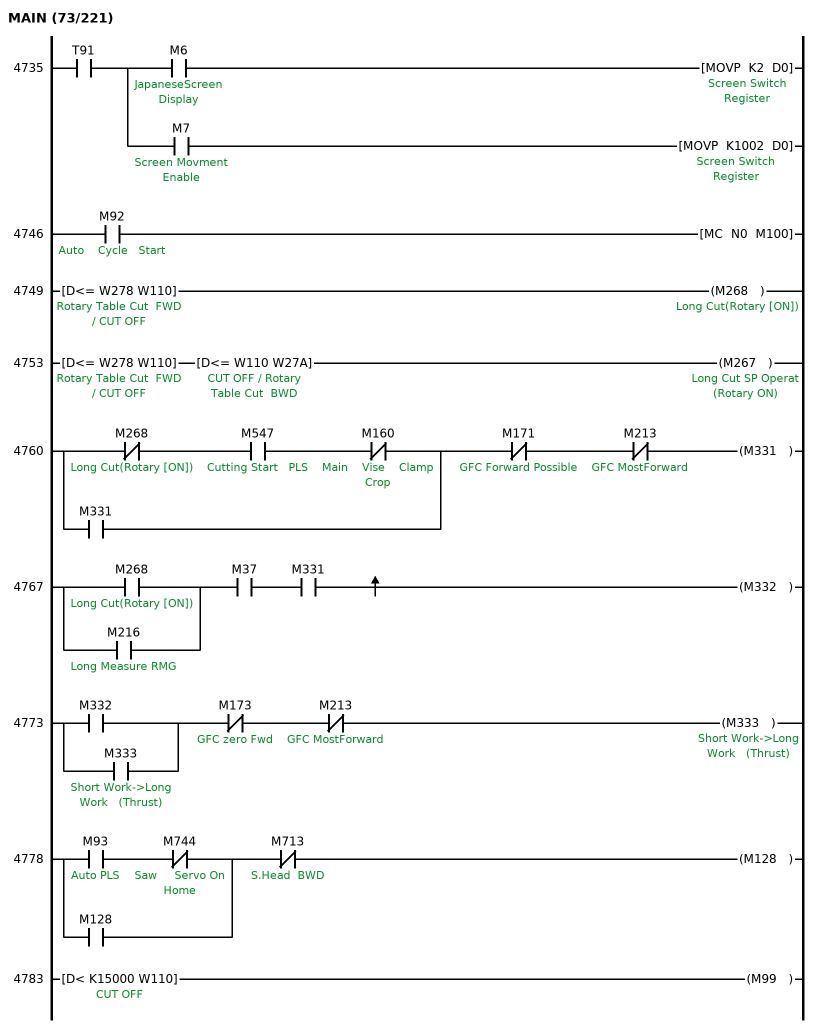
[picture p72: ladder of MAIN, rungs at steps 4735 to 4783]
4735  LD      T91
      MPS
      AND     M6  ; JapaneseScreen Display
      MOVP    K2 D0
      MPP
      AND     M7  ; Screen Movment Enable
      MOVP    K1002 D0
4746  LD      M92  ; Auto    Cycle   Start
      MC      N0 M100
4749  LDD<=   W278 W110  ; Rotary Table Cut  FWD / CUT OFF
      OUT     M268  ; Long Cut(Rotary [ON])
4753  LDD<=   W278 W110  ; Rotary Table Cut  FWD / CUT OFF
      ANDD<=  W110 W27A  ; CUT OFF / Rotary Table Cut  BWD
      OUT     M267  ; Long Cut SP Operat (Rotary ON)
4760  LDI     M268  ; Long Cut(Rotary [ON])
      AND     M547  ; Cutting Start   PLS
      ANI     M160  ; Main    Vise    Clamp   Crop
      OR      M331
      ANI     M171  ; GFC Forward Possible
      ANI     M213  ; GFC MostForward
      OUT     M331
4767  LD      M268  ; Long Cut(Rotary [ON])
      OR      M216  ; Long Measure RMG
      AND     M37
      AND     M331
      MEP
      OUT     M332
4773  LD      M332
      OR      M333  ; Short Work->Long Work   (Thrust)
      ANI     M173  ; GFC zero Fwd
      ANI     M213  ; GFC MostForward
      OUT     M333  ; Short Work->Long Work   (Thrust)
4778  LD      M93  ; Auto PLS
      ANI     M744  ; Saw     Servo On Home
      OR      M128
      ANI     M713  ; S.Head  BWD
      OUT     M128
4783  LDD<    K15000 W110  ; CUT OFF
      OUT     M99
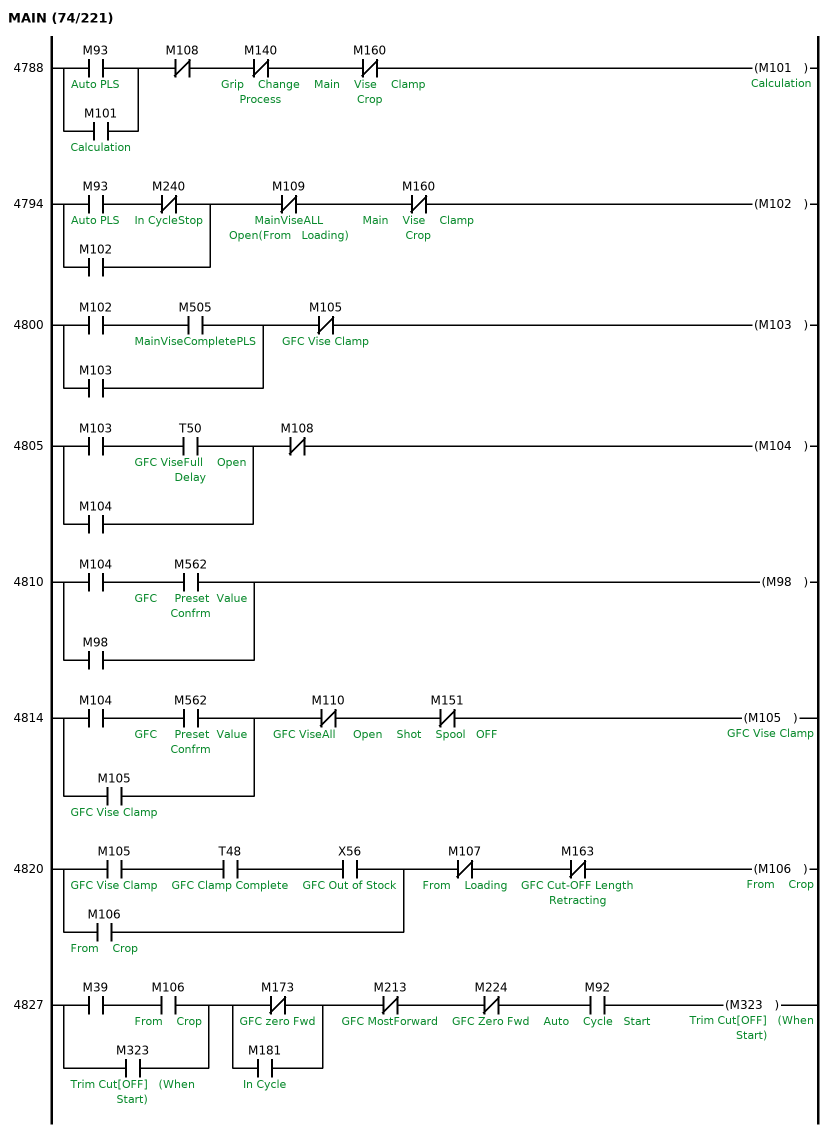
4788  LD      M93  ; Auto PLS
      OR      M101  ; Calculation
      ANI     M108
      ANI     M140  ; Grip    Change  Process
      ANI     M160  ; Main    Vise    Clamp   Crop
      OUT     M101  ; Calculation
4794  LD      M93  ; Auto PLS
      ANI     M240  ; In CycleStop
      OR      M102
      ANI     M109  ; MainViseALL Open(From   Loading)
      ANI     M160  ; Main    Vise    Clamp   Crop
      OUT     M102
4800  LD      M102
      AND     M505  ; MainViseCompletePLS
      OR      M103
      ANI     M105  ; GFC Vise Clamp
      OUT     M103
4805  LD      M103
      AND     T50  ; GFC ViseFull    Open    Delay
      OR      M104
      ANI     M108
      OUT     M104
4810  LD      M104
      AND     M562  ; GFC     Preset  Value   Confrm
      OR      M98
      OUT     M98
4814  LD      M104
      AND     M562  ; GFC     Preset  Value   Confrm
      OR      M105  ; GFC Vise Clamp
      ANI     M110  ; GFC ViseAll     Open
      ANI     M151  ; Shot    Spool   OFF
      OUT     M105  ; GFC Vise Clamp
4820  LD      M105  ; GFC Vise Clamp
      AND     T48  ; GFC Clamp Complete
      AND     X56  ; GFC Out of Stock
      OR      M106  ; From    Crop
      ANI     M107  ; From    Loading
      ANI     M163  ; GFC Cut-OFF Length Retracting
      OUT     M106  ; From    Crop
4827  LD      M39
      AND     M106  ; From    Crop
      OR      M323  ; Trim Cut[OFF]   (When   Start)
      LDI     M173  ; GFC zero Fwd
      OR      M181  ; In Cycle
      ANB
      ANI     M213  ; GFC MostForward
      ANI     M224  ; GFC Zero Fwd
      AND     M92  ; Auto    Cycle   Start
      OUT     M323  ; Trim Cut[OFF]   (When   Start)
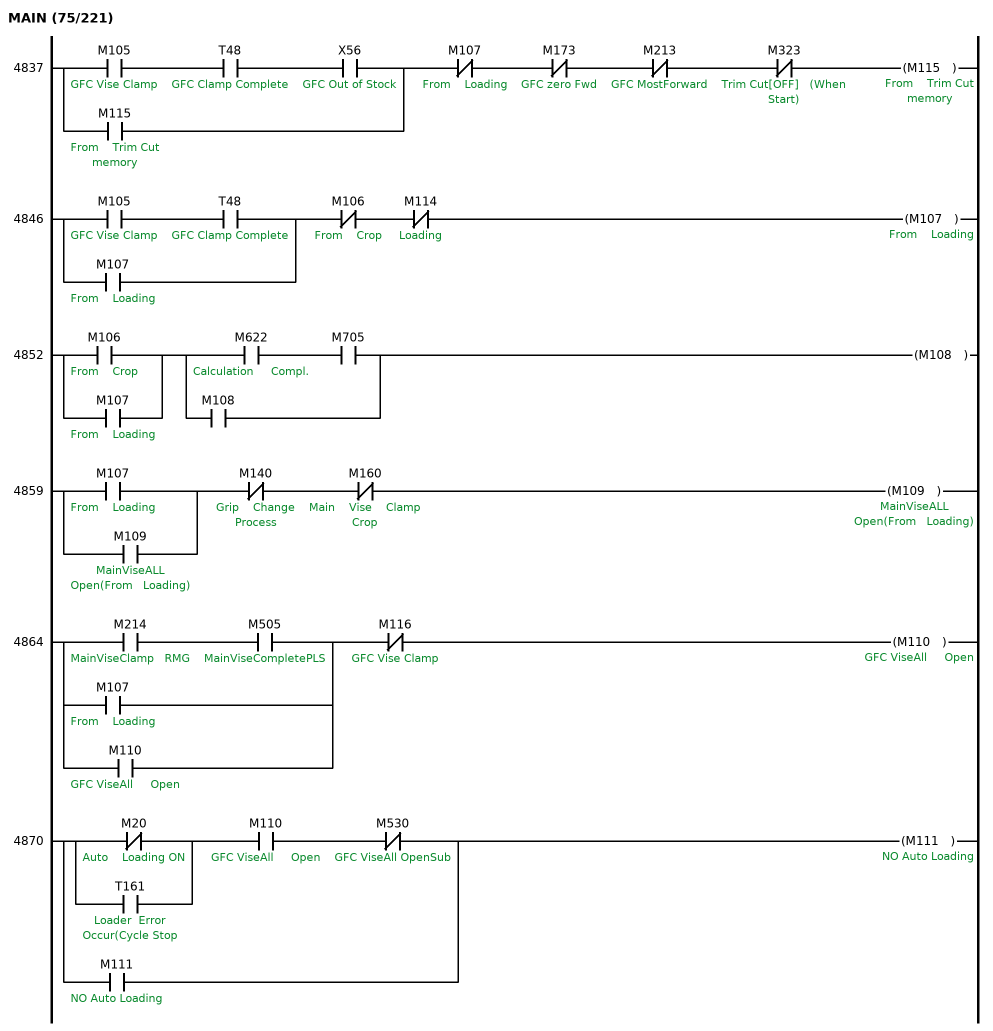
4837  LD      M105  ; GFC Vise Clamp
      AND     T48  ; GFC Clamp Complete
      AND     X56  ; GFC Out of Stock
      OR      M115  ; From    Trim Cut memory
      ANI     M107  ; From    Loading
      ANI     M173  ; GFC zero Fwd
      ANI     M213  ; GFC MostForward
      ANI     M323  ; Trim Cut[OFF]   (When   Start)
      OUT     M115  ; From    Trim Cut memory
4846  LD      M105  ; GFC Vise Clamp
      AND     T48  ; GFC Clamp Complete
      OR      M107  ; From    Loading
      ANI     M106  ; From    Crop
      ANI     M114  ; Loading
      OUT     M107  ; From    Loading
4852  LD      M106  ; From    Crop
      OR      M107  ; From    Loading
      LD      M622  ; Calculation     Compl.
      AND     M705
      OR      M108
      ANB
      OUT     M108
4859  LD      M107  ; From    Loading
      OR      M109  ; MainViseALL Open(From   Loading)
      ANI     M140  ; Grip    Change  Process
      ANI     M160  ; Main    Vise    Clamp   Crop
      OUT     M109  ; MainViseALL Open(From   Loading)
4864  LD      M214  ; MainViseClamp   RMG
      AND     M505  ; MainViseCompletePLS
      OR      M107  ; From    Loading
      OR      M110  ; GFC ViseAll     Open
      ANI     M116  ; GFC Vise Clamp
      OUT     M110  ; GFC ViseAll     Open
4870  LDI     M20  ; Auto    Loading ON
      OR      T161  ; Loader  Error   Occur(Cycle Stop
      AND     M110  ; GFC ViseAll     Open
      ANI     M530  ; GFC ViseAll OpenSub
      OR      M111  ; NO Auto Loading
      OUT     M111  ; NO Auto Loading
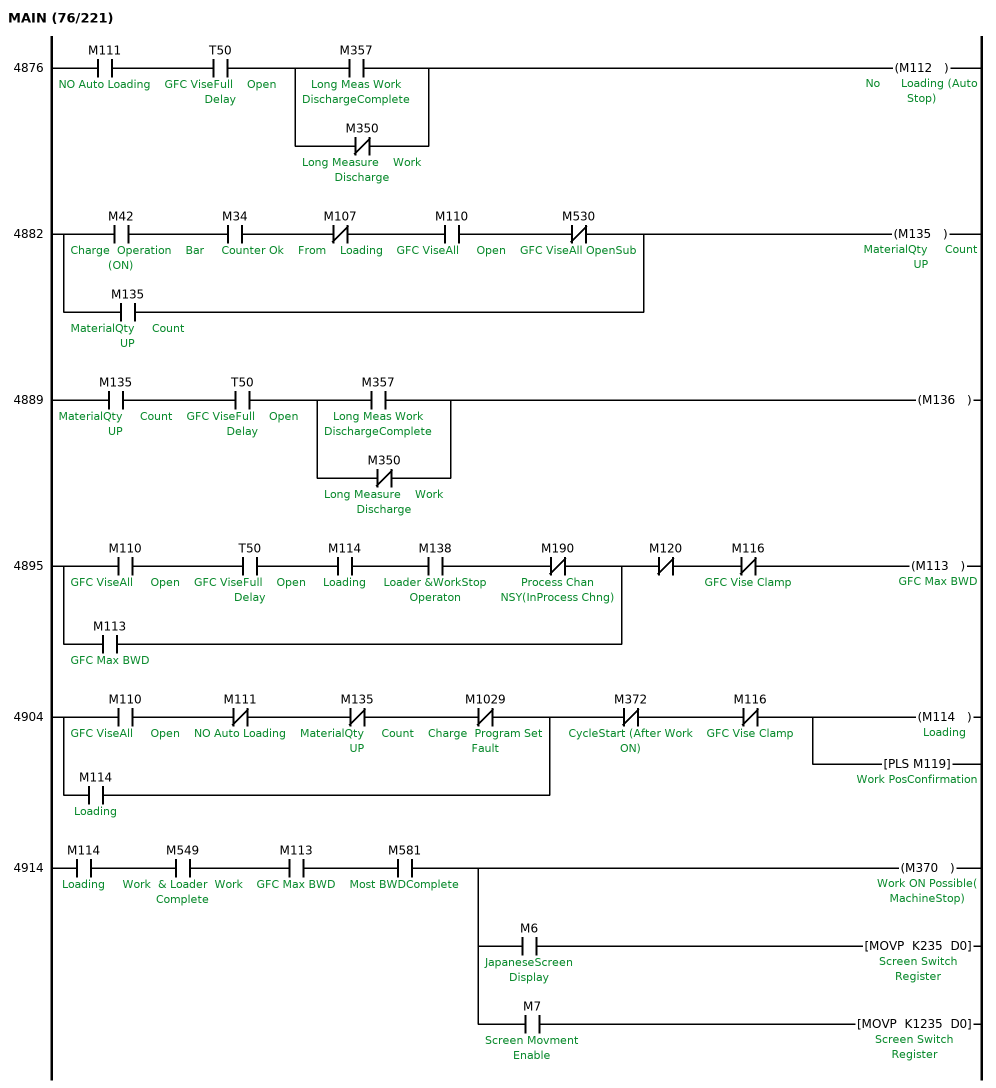
4876  LD      M111  ; NO Auto Loading
      AND     T50  ; GFC ViseFull    Open    Delay
      LD      M357  ; Long Meas Work DischargeComplete
      ORI     M350  ; Long Measure    Work Discharge
      ANB
      OUT     M112  ; No      Loading (Auto   Stop)
4882  LD      M42  ; Charge  Operation (ON)
      AND     M34  ; Bar     Counter Ok
      ANI     M107  ; From    Loading
      AND     M110  ; GFC ViseAll     Open
      ANI     M530  ; GFC ViseAll OpenSub
      OR      M135  ; MaterialQty     Count UP
      OUT     M135  ; MaterialQty     Count UP
4889  LD      M135  ; MaterialQty     Count UP
      AND     T50  ; GFC ViseFull    Open    Delay
      LD      M357  ; Long Meas Work DischargeComplete
      ORI     M350  ; Long Measure    Work Discharge
      ANB
      OUT     M136
4895  LD      M110  ; GFC ViseAll     Open
      AND     T50  ; GFC ViseFull    Open    Delay
      AND     M114  ; Loading
      AND     M138  ; Loader &WorkStopOperaton
      ANI     M190  ; Process Chan NSY(InProcess Chng)
      OR      M113  ; GFC Max BWD
      ANI     M120
      ANI     M116  ; GFC Vise Clamp
      OUT     M113  ; GFC Max BWD
4904  LD      M110  ; GFC ViseAll     Open
      ANI     M111  ; NO Auto Loading
      ANI     M135  ; MaterialQty     Count UP
      ANI     M1029  ; Charge  Program Set     Fault
      OR      M114  ; Loading
      ANI     M372  ; CycleStart (After Work ON)
      ANI     M116  ; GFC Vise Clamp
      OUT     M114  ; Loading
      PLS     M119  ; Work PosConfirmation
4914  LD      M114  ; Loading
      AND     M549  ; Work  & Loader  Work Complete
      AND     M113  ; GFC Max BWD
      AND     M581  ; Most BWDComplete
      OUT     M370  ; Work ON Possible(MachineStop)
      MPS
      AND     M6  ; JapaneseScreen Display
      MOVP    K235 D0
      MPP
      AND     M7  ; Screen Movment Enable
      MOVP    K1235 D0
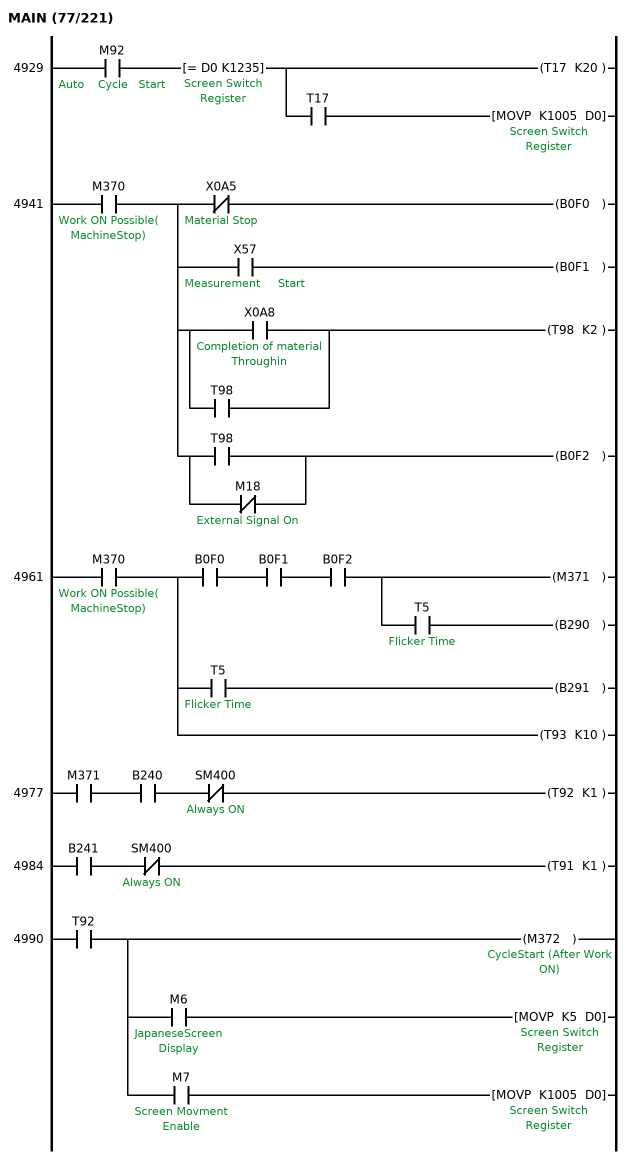
4929  LD      M92  ; Auto    Cycle   Start
      AND=    D0 K1235  ; Screen Switch Register
      OUT     T17 K20
      AND     T17
      MOVP    K1005 D0
4941  LD      M370  ; Work ON Possible(MachineStop)
      MPS
      ANI     X0A5  ; Material Stop
      OUT     B0F0
      MRD
      AND     X57  ; Measurement     Start
      OUT     B0F1
      MRD
      LD      X0A8  ; Completion of material Throughin
      OR      T98
      ANB
      OUT     T98 K2
      MPP
      LD      T98
      ORI     M18  ; External Signal On
      ANB
      OUT     B0F2
4961  LD      M370  ; Work ON Possible(MachineStop)
      MPS
      AND     B0F0
      AND     B0F1
      AND     B0F2
      OUT     M371
      AND     T5  ; Flicker Time
      OUT     B290
      MRD
      AND     T5  ; Flicker Time
      OUT     B291
      MPP
      OUT     T93 K10
4977  LD      M371
      AND     B240
      ANI     SM400  ; Always ON
      OUT     T92 K1
4984  LD      B241
      ANI     SM400  ; Always ON
      OUT     T91 K1
4990  LD      T92
      OUT     M372  ; CycleStart (After Work ON)
      MPS
      AND     M6  ; JapaneseScreen Display
      MOVP    K5 D0
      MPP
      AND     M7  ; Screen Movment Enable
      MOVP    K1005 D0
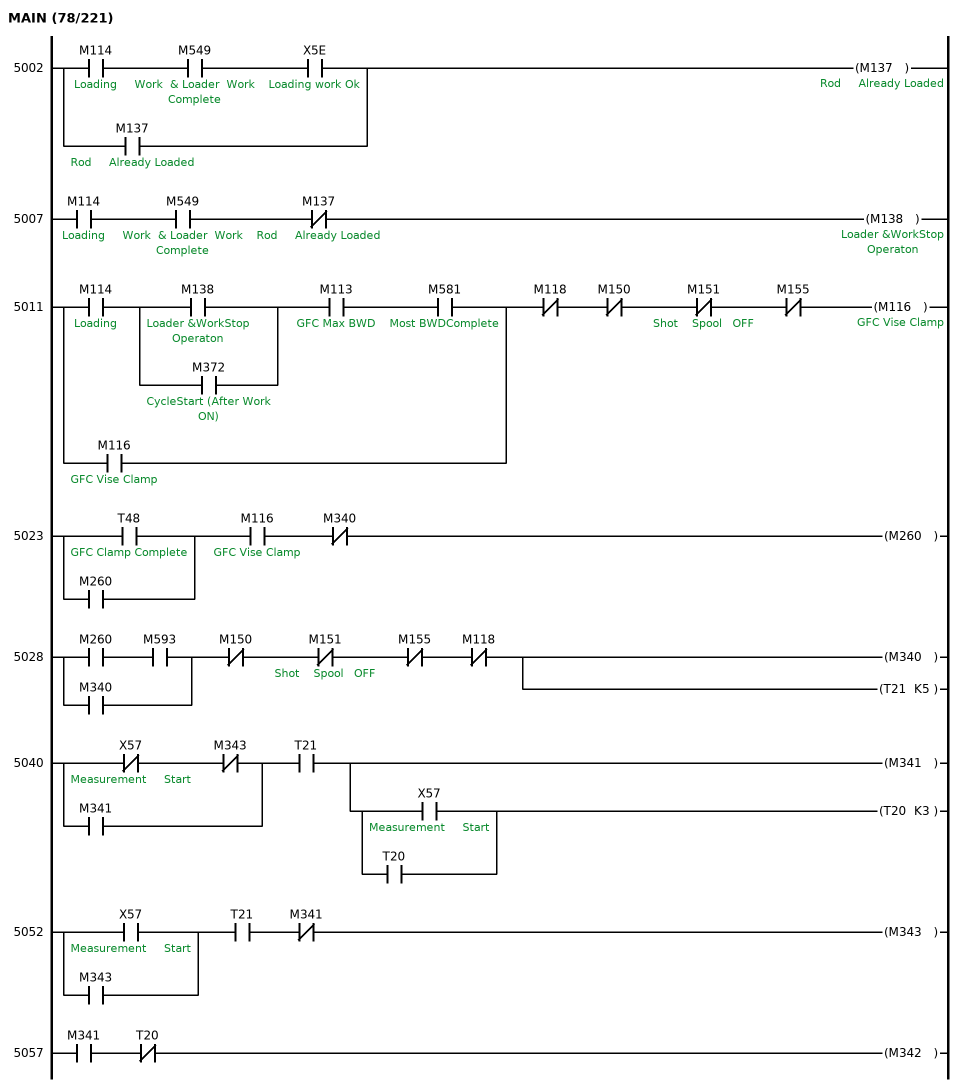
5002  LD      M114  ; Loading
      AND     M549  ; Work  & Loader  Work Complete
      AND     X5E  ; Loading work Ok
      OR      M137  ; Rod     Already Loaded
      OUT     M137  ; Rod     Already Loaded
5007  LD      M114  ; Loading
      AND     M549  ; Work  & Loader  Work Complete
      ANI     M137  ; Rod     Already Loaded
      OUT     M138  ; Loader &WorkStopOperaton
5011  LD      M114  ; Loading
      LD      M138  ; Loader &WorkStopOperaton
      OR      M372  ; CycleStart (After Work ON)
      ANB
      AND     M113  ; GFC Max BWD
      AND     M581  ; Most BWDComplete
      OR      M116  ; GFC Vise Clamp
      ANI     M118
      ANI     M150
      ANI     M151  ; Shot    Spool   OFF
      ANI     M155
      OUT     M116  ; GFC Vise Clamp
5023  LD      T48  ; GFC Clamp Complete
      OR      M260
      AND     M116  ; GFC Vise Clamp
      ANI     M340
      OUT     M260
5028  LD      M260
      AND     M593
      OR      M340
      ANI     M150
      ANI     M151  ; Shot    Spool   OFF
      ANI     M155
      ANI     M118
      OUT     M340
      OUT     T21 K5
5040  LDI     X57  ; Measurement     Start
      ANI     M343
      OR      M341
      AND     T21
      OUT     M341
      LD      X57  ; Measurement     Start
      OR      T20
      ANB
      OUT     T20 K3
5052  LD      X57  ; Measurement     Start
      OR      M343
      AND     T21
      ANI     M341
      OUT     M343
5057  LD      M341
      ANI     T20
      OUT     M342
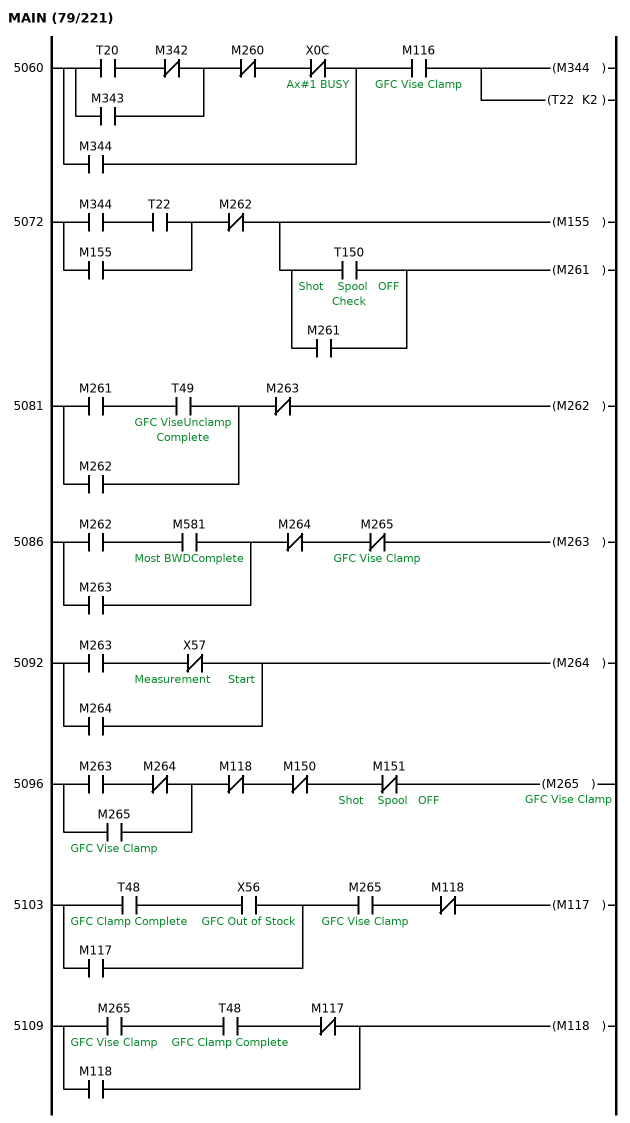
5060  LD      T20
      ANI     M342
      OR      M343
      ANI     M260
      ANI     X0C  ; Ax#1 BUSY
      OR      M344
      AND     M116  ; GFC Vise Clamp
      OUT     M344
      OUT     T22 K2
5072  LD      M344
      AND     T22
      OR      M155
      ANI     M262
      OUT     M155
      LD      T150  ; Shot    Spool   OFF     Check
      OR      M261
      ANB
      OUT     M261
5081  LD      M261
      AND     T49  ; GFC ViseUnclamp Complete
      OR      M262
      ANI     M263
      OUT     M262
5086  LD      M262
      AND     M581  ; Most BWDComplete
      OR      M263
      ANI     M264
      ANI     M265  ; GFC Vise Clamp
      OUT     M263
5092  LD      M263
      ANI     X57  ; Measurement     Start
      OR      M264
      OUT     M264
5096  LD      M263
      ANI     M264
      OR      M265  ; GFC Vise Clamp
      ANI     M118
      ANI     M150
      ANI     M151  ; Shot    Spool   OFF
      OUT     M265  ; GFC Vise Clamp
5103  LD      T48  ; GFC Clamp Complete
      AND     X56  ; GFC Out of Stock
      OR      M117
      AND     M265  ; GFC Vise Clamp
      ANI     M118
      OUT     M117
5109  LD      M265  ; GFC Vise Clamp
      AND     T48  ; GFC Clamp Complete
      ANI     M117
      OR      M118
      OUT     M118
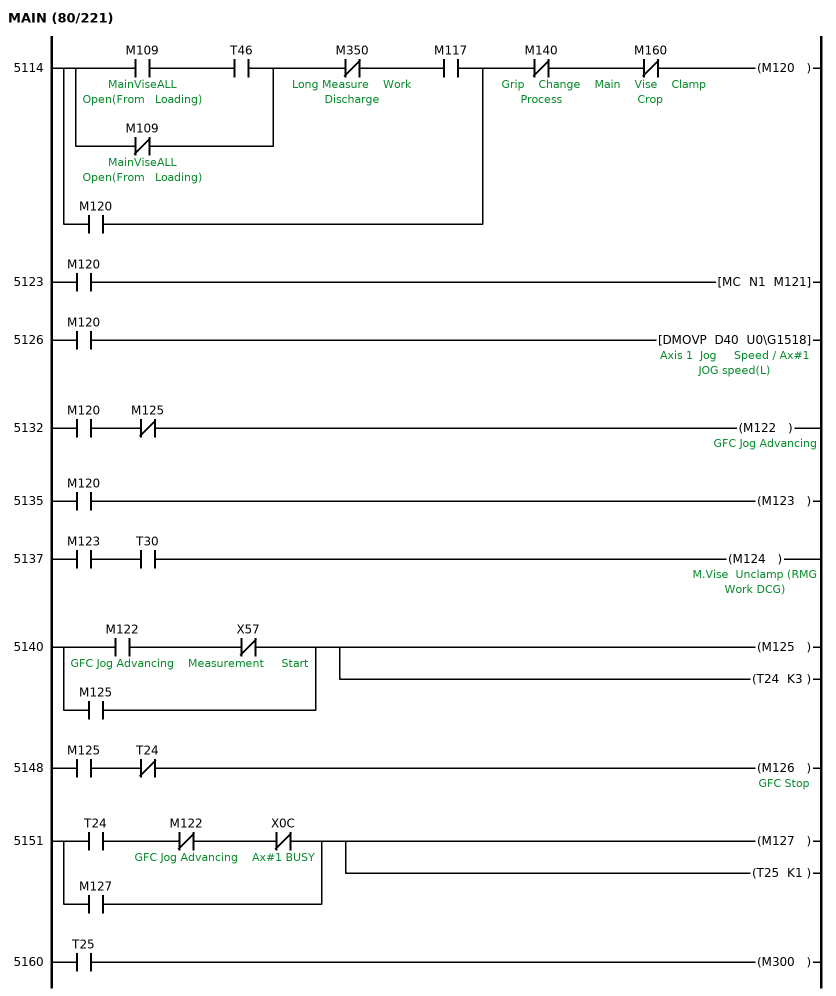
5114  LD      M109  ; MainViseALL Open(From   Loading)
      AND     T46
      ORI     M109  ; MainViseALL Open(From   Loading)
      ANI     M350  ; Long Measure    Work Discharge
      AND     M117
      OR      M120
      ANI     M140  ; Grip    Change  Process
      ANI     M160  ; Main    Vise    Clamp   Crop
      OUT     M120
5123  LD      M120
      MC      N1 M121
5126  LD      M120
      DMOVP   D40 U0\G1518
5132  LD      M120
      ANI     M125
      OUT     M122  ; GFC Jog Advancing
5135  LD      M120
      OUT     M123
5137  LD      M123
      AND     T30
      OUT     M124  ; M.Vise  Unclamp (RMG Work DCG)
5140  LD      M122  ; GFC Jog Advancing
      ANI     X57  ; Measurement     Start
      OR      M125
      OUT     M125
      OUT     T24 K3
5148  LD      M125
      ANI     T24
      OUT     M126  ; GFC Stop
5151  LD      T24
      ANI     M122  ; GFC Jog Advancing
      ANI     X0C  ; Ax#1 BUSY
      OR      M127
      OUT     M127
      OUT     T25 K1
5160  LD      T25
      OUT     M300
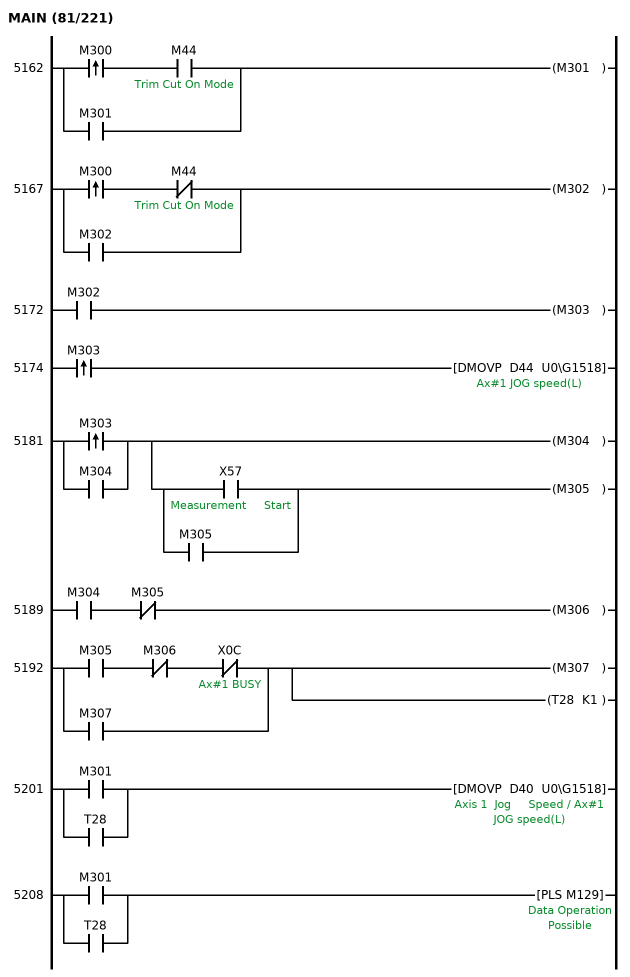
5162  LDP     M300
      AND     M44  ; Trim Cut On Mode
      OR      M301
      OUT     M301
5167  LDP     M300
      ANI     M44  ; Trim Cut On Mode
      OR      M302
      OUT     M302
5172  LD      M302
      OUT     M303
5174  LDP     M303
      DMOVP   D44 U0\G1518
5181  LDP     M303
      OR      M304
      OUT     M304
      LD      X57  ; Measurement     Start
      OR      M305
      ANB
      OUT     M305
5189  LD      M304
      ANI     M305
      OUT     M306
5192  LD      M305
      ANI     M306
      ANI     X0C  ; Ax#1 BUSY
      OR      M307
      OUT     M307
      OUT     T28 K1
5201  LD      M301
      OR      T28
      DMOVP   D40 U0\G1518
5208  LD      M301
      OR      T28
      PLS     M129  ; Data Operation  Possible
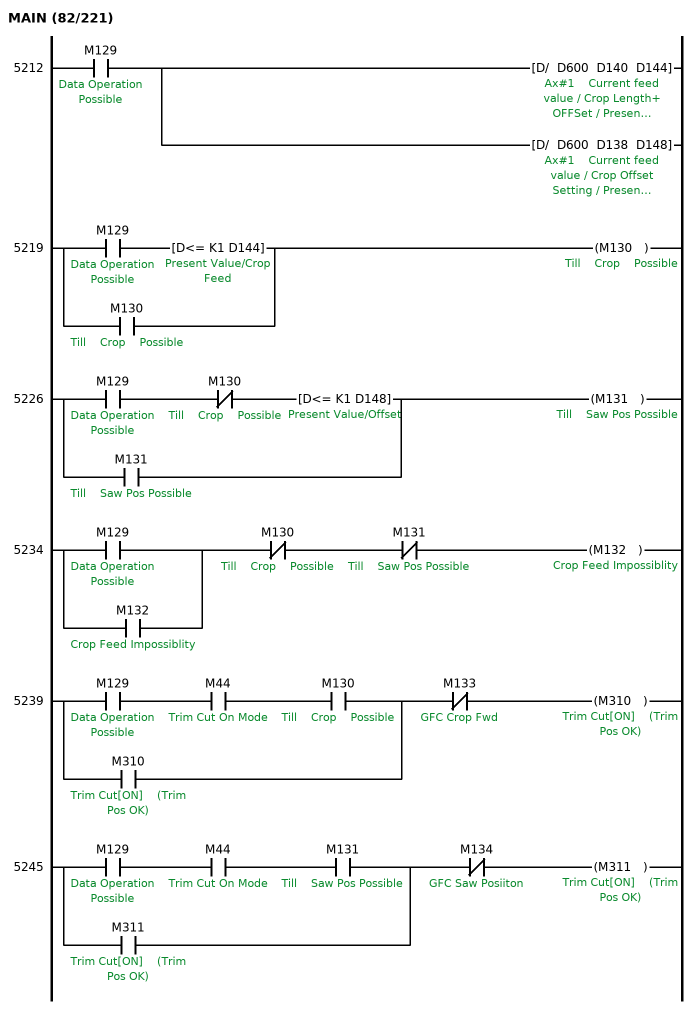
5212  LD      M129  ; Data Operation  Possible
      D/      D600 D140 D144  ; Crop Length+ OFFSet / Present Value/Crop Feed
      D/      D600 D138 D148  ; Crop Offset Setting / Present Value/Offset
5219  LD      M129  ; Data Operation  Possible
      ANDD<=  K1 D144  ; Present Value/Crop Feed
      OR      M130  ; Till    Crop    Possible
      OUT     M130  ; Till    Crop    Possible
5226  LD      M129  ; Data Operation  Possible
      ANI     M130  ; Till    Crop    Possible
      ANDD<=  K1 D148  ; Present Value/Offset
      OR      M131  ; Till    Saw Pos Possible
      OUT     M131  ; Till    Saw Pos Possible
5234  LD      M129  ; Data Operation  Possible
      OR      M132  ; Crop Feed Impossiblity
      ANI     M130  ; Till    Crop    Possible
      ANI     M131  ; Till    Saw Pos Possible
      OUT     M132  ; Crop Feed Impossiblity
5239  LD      M129  ; Data Operation  Possible
      AND     M44  ; Trim Cut On Mode
      AND     M130  ; Till    Crop    Possible
      OR      M310  ; Trim Cut[ON]    (Trim Pos OK)
      ANI     M133  ; GFC Crop Fwd
      OUT     M310  ; Trim Cut[ON]    (Trim Pos OK)
5245  LD      M129  ; Data Operation  Possible
      AND     M44  ; Trim Cut On Mode
      AND     M131  ; Till    Saw Pos Possible
      OR      M311  ; Trim Cut[ON]    (Trim Pos OK)
      ANI     M134  ; GFC Saw Posiiton
      OUT     M311  ; Trim Cut[ON]    (Trim Pos OK)
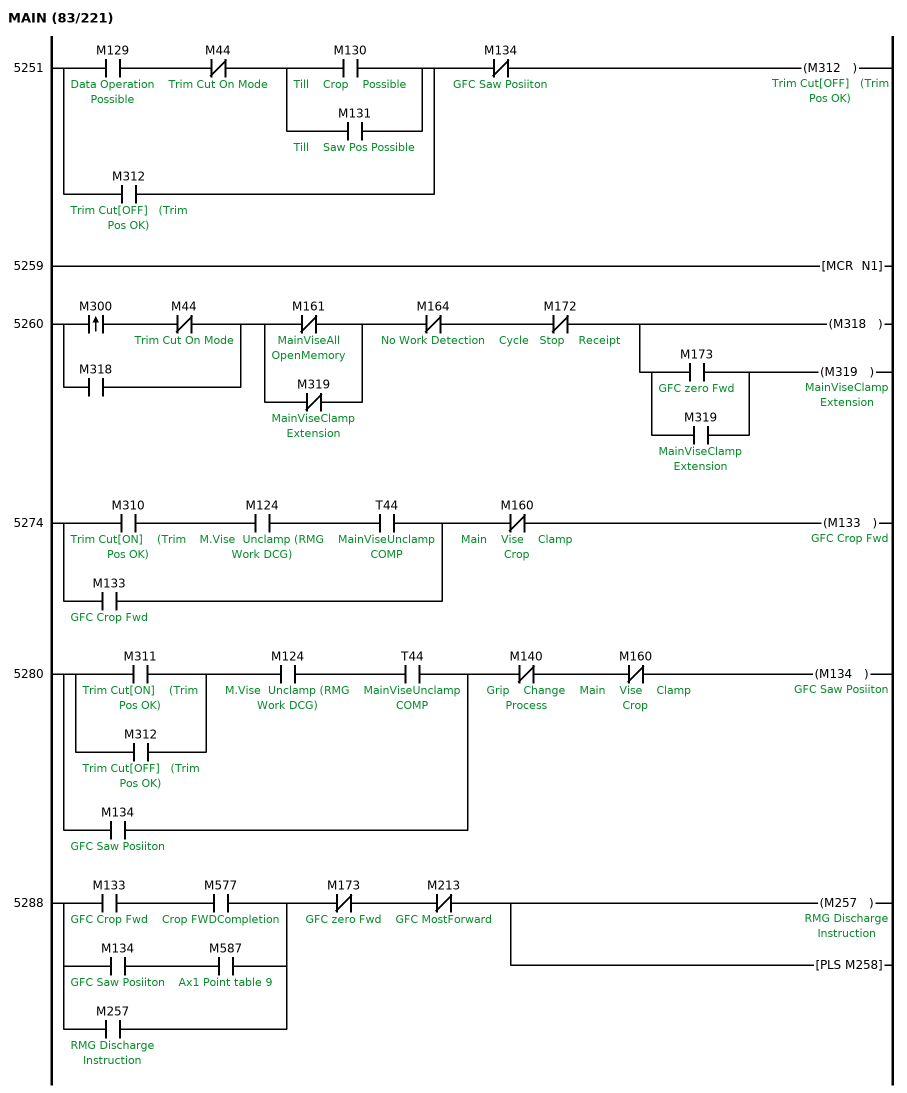
5251  LD      M129  ; Data Operation  Possible
      ANI     M44  ; Trim Cut On Mode
      LD      M130  ; Till    Crop    Possible
      OR      M131  ; Till    Saw Pos Possible
      ANB
      OR      M312  ; Trim Cut[OFF]   (Trim Pos OK)
      ANI     M134  ; GFC Saw Posiiton
      OUT     M312  ; Trim Cut[OFF]   (Trim Pos OK)
5259  MCR     N1
5260  LDP     M300
      ANI     M44  ; Trim Cut On Mode
      OR      M318
      LDI     M161  ; MainViseAll OpenMemory
      ORI     M319  ; MainViseClamp   Extension
      ANB
      ANI     M164  ; No Work Detection
      ANI     M172  ; Cycle   Stop    Receipt
      OUT     M318
      LD      M173  ; GFC zero Fwd
      OR      M319  ; MainViseClamp   Extension
      ANB
      OUT     M319  ; MainViseClamp   Extension
5274  LD      M310  ; Trim Cut[ON]    (Trim Pos OK)
      AND     M124  ; M.Vise  Unclamp (RMG Work DCG)
      AND     T44  ; MainViseUnclamp COMP
      OR      M133  ; GFC Crop Fwd
      ANI     M160  ; Main    Vise    Clamp   Crop
      OUT     M133  ; GFC Crop Fwd
5280  LD      M311  ; Trim Cut[ON]    (Trim Pos OK)
      OR      M312  ; Trim Cut[OFF]   (Trim Pos OK)
      AND     M124  ; M.Vise  Unclamp (RMG Work DCG)
      AND     T44  ; MainViseUnclamp COMP
      OR      M134  ; GFC Saw Posiiton
      ANI     M140  ; Grip    Change  Process
      ANI     M160  ; Main    Vise    Clamp   Crop
      OUT     M134  ; GFC Saw Posiiton
5288  LD      M133  ; GFC Crop Fwd
      AND     M577  ; Crop FWDCompletion
      LD      M134  ; GFC Saw Posiiton
      AND     M587  ; Ax1 Point table 9
      ORB
      OR      M257  ; RMG Discharge Instruction
      ANI     M173  ; GFC zero Fwd
      ANI     M213  ; GFC MostForward
      OUT     M257  ; RMG Discharge Instruction
      PLS     M258
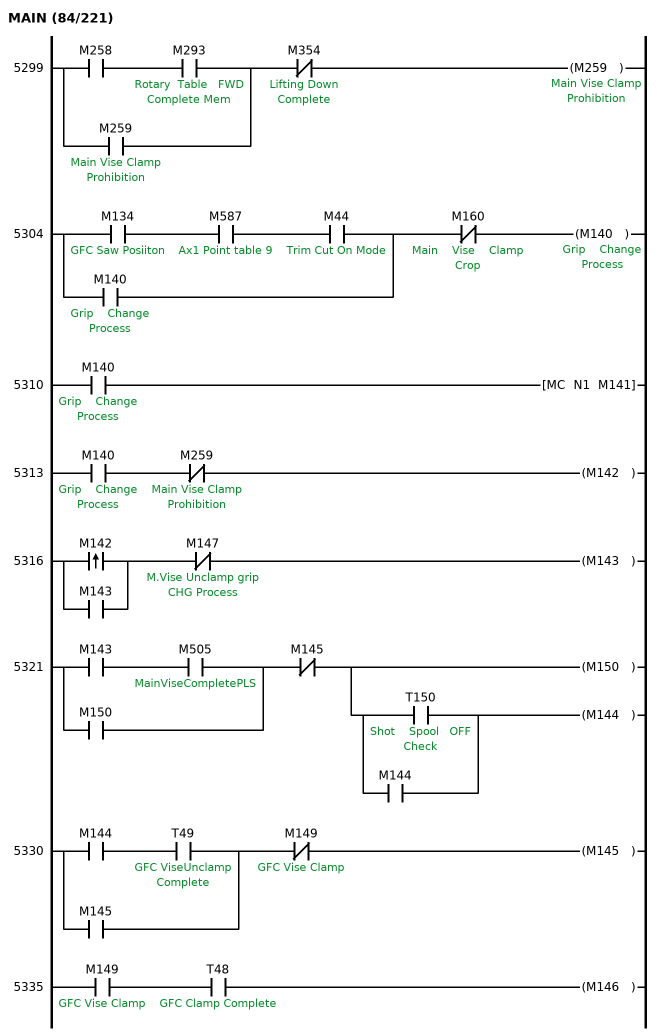
5299  LD      M258
      AND     M293  ; Rotary  Table   FWD Complete Mem
      OR      M259  ; Main Vise Clamp Prohibition
      ANI     M354  ; Lifting Down    Complete
      OUT     M259  ; Main Vise Clamp Prohibition
5304  LD      M134  ; GFC Saw Posiiton
      AND     M587  ; Ax1 Point table 9
      AND     M44  ; Trim Cut On Mode
      OR      M140  ; Grip    Change  Process
      ANI     M160  ; Main    Vise    Clamp   Crop
      OUT     M140  ; Grip    Change  Process
5310  LD      M140  ; Grip    Change  Process
      MC      N1 M141
5313  LD      M140  ; Grip    Change  Process
      ANI     M259  ; Main Vise Clamp Prohibition
      OUT     M142
5316  LDP     M142
      OR      M143
      ANI     M147  ; M.Vise Unclamp grip CHG Process
      OUT     M143
5321  LD      M143
      AND     M505  ; MainViseCompletePLS
      OR      M150
      ANI     M145
      OUT     M150
      LD      T150  ; Shot    Spool   OFF     Check
      OR      M144
      ANB
      OUT     M144
5330  LD      M144
      AND     T49  ; GFC ViseUnclamp Complete
      OR      M145
      ANI     M149  ; GFC Vise Clamp
      OUT     M145
5335  LD      M149  ; GFC Vise Clamp
      AND     T48  ; GFC Clamp Complete
      OUT     M146
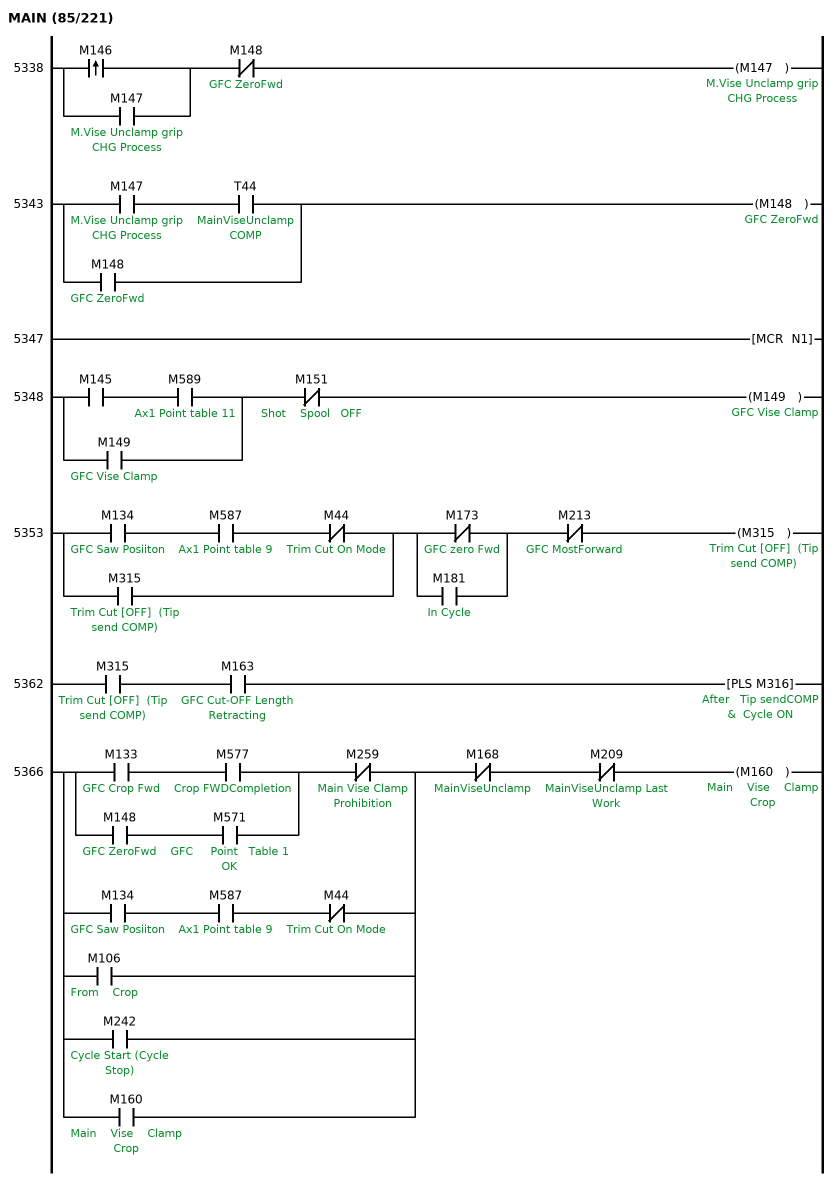
5338  LDP     M146
      OR      M147  ; M.Vise Unclamp grip CHG Process
      ANI     M148  ; GFC ZeroFwd
      OUT     M147  ; M.Vise Unclamp grip CHG Process
5343  LD      M147  ; M.Vise Unclamp grip CHG Process
      AND     T44  ; MainViseUnclamp COMP
      OR      M148  ; GFC ZeroFwd
      OUT     M148  ; GFC ZeroFwd
5347  MCR     N1
5348  LD      M145
      AND     M589  ; Ax1 Point table 11
      OR      M149  ; GFC Vise Clamp
      ANI     M151  ; Shot    Spool   OFF
      OUT     M149  ; GFC Vise Clamp
5353  LD      M134  ; GFC Saw Posiiton
      AND     M587  ; Ax1 Point table 9
      ANI     M44  ; Trim Cut On Mode
      OR      M315  ; Trim Cut [OFF]  (Tip send COMP)
      LDI     M173  ; GFC zero Fwd
      OR      M181  ; In Cycle
      ANB
      ANI     M213  ; GFC MostForward
      OUT     M315  ; Trim Cut [OFF]  (Tip send COMP)
5362  LD      M315  ; Trim Cut [OFF]  (Tip send COMP)
      AND     M163  ; GFC Cut-OFF Length Retracting
      PLS     M316  ; After   Tip sendCOMP &  Cycle ON
5366  LD      M133  ; GFC Crop Fwd
      AND     M577  ; Crop FWDCompletion
      LD      M148  ; GFC ZeroFwd
      AND     M571  ; GFC     Point   Table 1 OK
      ORB
      ANI     M259  ; Main Vise Clamp Prohibition
      LD      M134  ; GFC Saw Posiiton
      AND     M587  ; Ax1 Point table 9
      ANI     M44  ; Trim Cut On Mode
      ORB
      OR      M106  ; From    Crop
      OR      M242  ; Cycle Start (Cycle Stop)
      OR      M160  ; Main    Vise    Clamp   Crop
      ANI     M168  ; MainViseUnclamp
      ANI     M209  ; MainViseUnclamp Last    Work
      OUT     M160  ; Main    Vise    Clamp   Crop
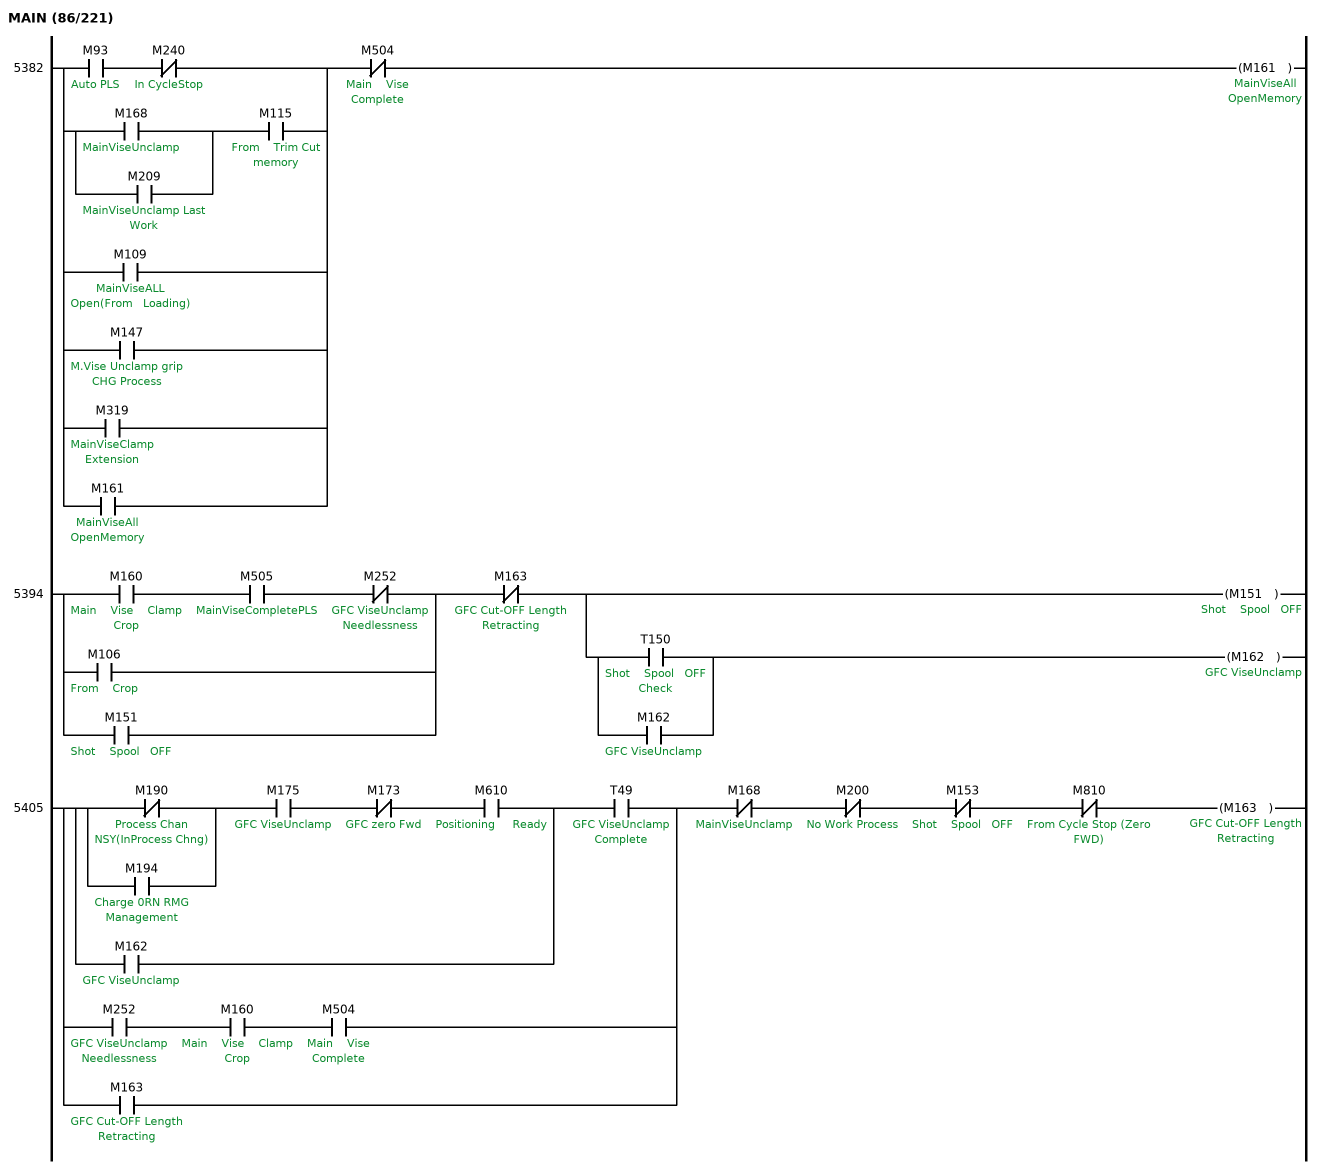
5382  LD      M93  ; Auto PLS
      ANI     M240  ; In CycleStop
      LD      M168  ; MainViseUnclamp
      OR      M209  ; MainViseUnclamp Last    Work
      AND     M115  ; From    Trim Cut memory
      ORB
      OR      M109  ; MainViseALL Open(From   Loading)
      OR      M147  ; M.Vise Unclamp grip CHG Process
      OR      M319  ; MainViseClamp   Extension
      OR      M161  ; MainViseAll OpenMemory
      ANI     M504  ; Main    Vise    Complete
      OUT     M161  ; MainViseAll OpenMemory
5394  LD      M160  ; Main    Vise    Clamp   Crop
      AND     M505  ; MainViseCompletePLS
      ANI     M252  ; GFC ViseUnclamp Needlessness
      OR      M106  ; From    Crop
      OR      M151  ; Shot    Spool   OFF
      ANI     M163  ; GFC Cut-OFF Length Retracting
      OUT     M151  ; Shot    Spool   OFF
      LD      T150  ; Shot    Spool   OFF     Check
      OR      M162  ; GFC ViseUnclamp
      ANB
      OUT     M162  ; GFC ViseUnclamp
5405  LDI     M190  ; Process Chan NSY(InProcess Chng)
      OR      M194  ; Charge 0RN RMG  Management
      AND     M175  ; GFC ViseUnclamp
      ANI     M173  ; GFC zero Fwd
      AND     M610  ; Positioning     Ready
      OR      M162  ; GFC ViseUnclamp
      AND     T49  ; GFC ViseUnclamp Complete
      LD      M252  ; GFC ViseUnclamp Needlessness
      AND     M160  ; Main    Vise    Clamp   Crop
      AND     M504  ; Main    Vise    Complete
      ORB
      OR      M163  ; GFC Cut-OFF Length Retracting
      ANI     M168  ; MainViseUnclamp
      ANI     M200  ; No Work Process
      ANI     M153  ; Shot    Spool   OFF
      ANI     M810  ; From Cycle Stop (Zero   FWD)
      OUT     M163  ; GFC Cut-OFF Length Retracting
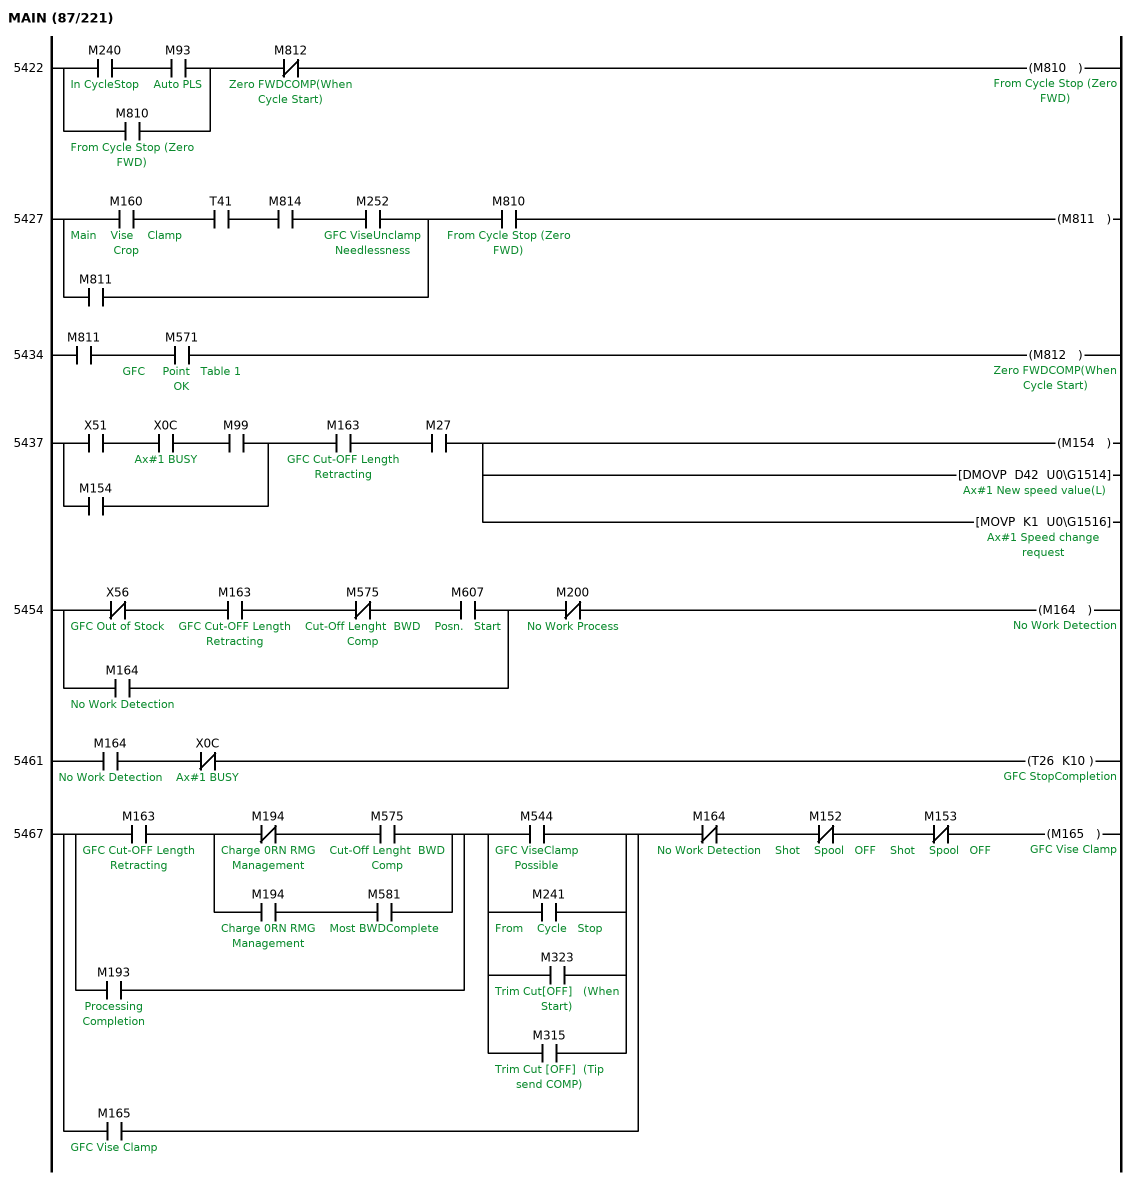
5422  LD      M240  ; In CycleStop
      AND     M93  ; Auto PLS
      OR      M810  ; From Cycle Stop (Zero   FWD)
      ANI     M812  ; Zero FWDCOMP(When Cycle Start)
      OUT     M810  ; From Cycle Stop (Zero   FWD)
5427  LD      M160  ; Main    Vise    Clamp   Crop
      AND     T41
      AND     M814
      AND     M252  ; GFC ViseUnclamp Needlessness
      OR      M811
      AND     M810  ; From Cycle Stop (Zero   FWD)
      OUT     M811
5434  LD      M811
      AND     M571  ; GFC     Point   Table 1 OK
      OUT     M812  ; Zero FWDCOMP(When Cycle Start)
5437  LD      X51
      AND     X0C  ; Ax#1 BUSY
      AND     M99
      OR      M154
      AND     M163  ; GFC Cut-OFF Length Retracting
      AND     M27
      OUT     M154
      DMOVP   D42 U0\G1514  ; Ax#1 New speed value(L)
      MOVP    K1 U0\G1516  ; Ax#1 Speed change request
5454  LDI     X56  ; GFC Out of Stock
      AND     M163  ; GFC Cut-OFF Length Retracting
      ANI     M575  ; Cut-Off Lenght  BWD Comp
      AND     M607  ; Posn.   Start
      OR      M164  ; No Work Detection
      ANI     M200  ; No Work Process
      OUT     M164  ; No Work Detection
5461  LD      M164  ; No Work Detection
      ANI     X0C  ; Ax#1 BUSY
      OUT     T26 K10  ; GFC StopCompletion
5467  LD      M163  ; GFC Cut-OFF Length Retracting
      LDI     M194  ; Charge 0RN RMG  Management
      AND     M575  ; Cut-Off Lenght  BWD Comp
      LD      M194  ; Charge 0RN RMG  Management
      AND     M581  ; Most BWDComplete
      ORB
      ANB
      OR      M193  ; Processing      Completion
      LD      M544  ; GFC ViseClamp   Possible
      OR      M241  ; From    Cycle   Stop
      OR      M323  ; Trim Cut[OFF]   (When   Start)
      OR      M315  ; Trim Cut [OFF]  (Tip send COMP)
      ANB
      OR      M165  ; GFC Vise Clamp
      ANI     M164  ; No Work Detection
      ANI     M152  ; Shot    Spool   OFF
      ANI     M153  ; Shot    Spool   OFF
      OUT     M165  ; GFC Vise Clamp
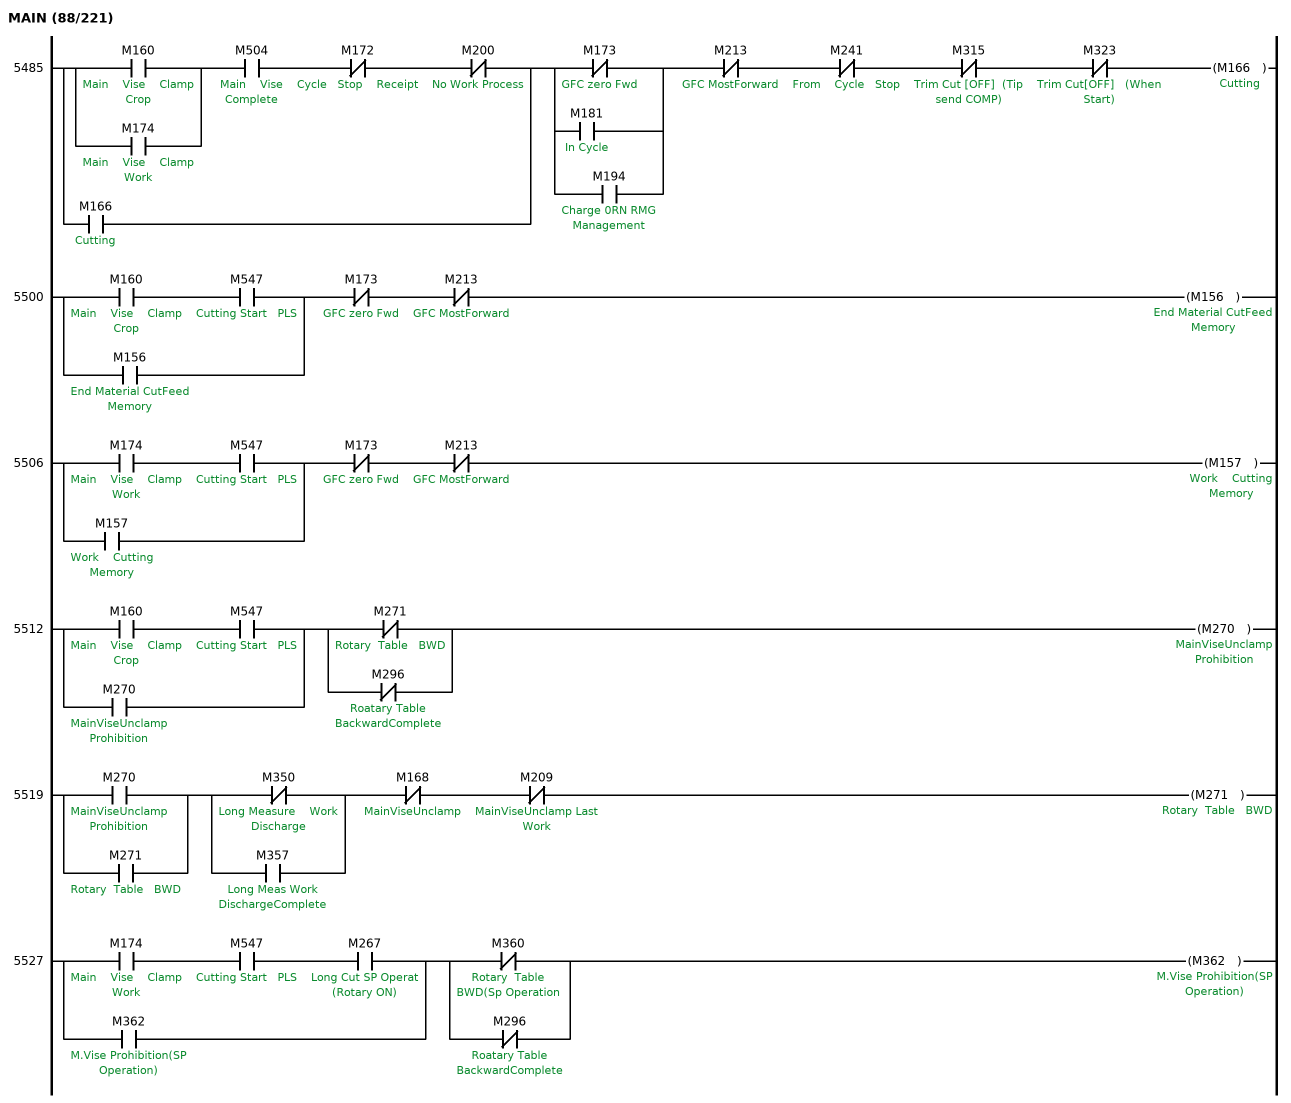
5485  LD      M160  ; Main    Vise    Clamp   Crop
      OR      M174  ; Main    Vise    Clamp   Work
      AND     M504  ; Main    Vise    Complete
      ANI     M172  ; Cycle   Stop    Receipt
      ANI     M200  ; No Work Process
      OR      M166  ; Cutting
      LDI     M173  ; GFC zero Fwd
      OR      M181  ; In Cycle
      OR      M194  ; Charge 0RN RMG  Management
      ANB
      ANI     M213  ; GFC MostForward
      ANI     M241  ; From    Cycle   Stop
      ANI     M315  ; Trim Cut [OFF]  (Tip send COMP)
      ANI     M323  ; Trim Cut[OFF]   (When   Start)
      OUT     M166  ; Cutting
5500  LD      M160  ; Main    Vise    Clamp   Crop
      AND     M547  ; Cutting Start   PLS
      OR      M156  ; End Material CutFeed Memory
      ANI     M173  ; GFC zero Fwd
      ANI     M213  ; GFC MostForward
      OUT     M156  ; End Material CutFeed Memory
5506  LD      M174  ; Main    Vise    Clamp   Work
      AND     M547  ; Cutting Start   PLS
      OR      M157  ; Work    Cutting Memory
      ANI     M173  ; GFC zero Fwd
      ANI     M213  ; GFC MostForward
      OUT     M157  ; Work    Cutting Memory
5512  LD      M160  ; Main    Vise    Clamp   Crop
      AND     M547  ; Cutting Start   PLS
      OR      M270  ; MainViseUnclamp Prohibition
      LDI     M271  ; Rotary  Table   BWD
      ORI     M296  ; Roatary Table   BackwardComplete
      ANB
      OUT     M270  ; MainViseUnclamp Prohibition
5519  LD      M270  ; MainViseUnclamp Prohibition
      OR      M271  ; Rotary  Table   BWD
      LDI     M350  ; Long Measure    Work Discharge
      OR      M357  ; Long Meas Work DischargeComplete
      ANB
      ANI     M168  ; MainViseUnclamp
      ANI     M209  ; MainViseUnclamp Last    Work
      OUT     M271  ; Rotary  Table   BWD
5527  LD      M174  ; Main    Vise    Clamp   Work
      AND     M547  ; Cutting Start   PLS
      AND     M267  ; Long Cut SP Operat (Rotary ON)
      OR      M362  ; M.Vise Prohibition(SP Operation)
      LDI     M360  ; Rotary  Table   BWD(Sp Operation
      ORI     M296  ; Roatary Table   BackwardComplete
      ANB
      OUT     M362  ; M.Vise Prohibition(SP Operation)
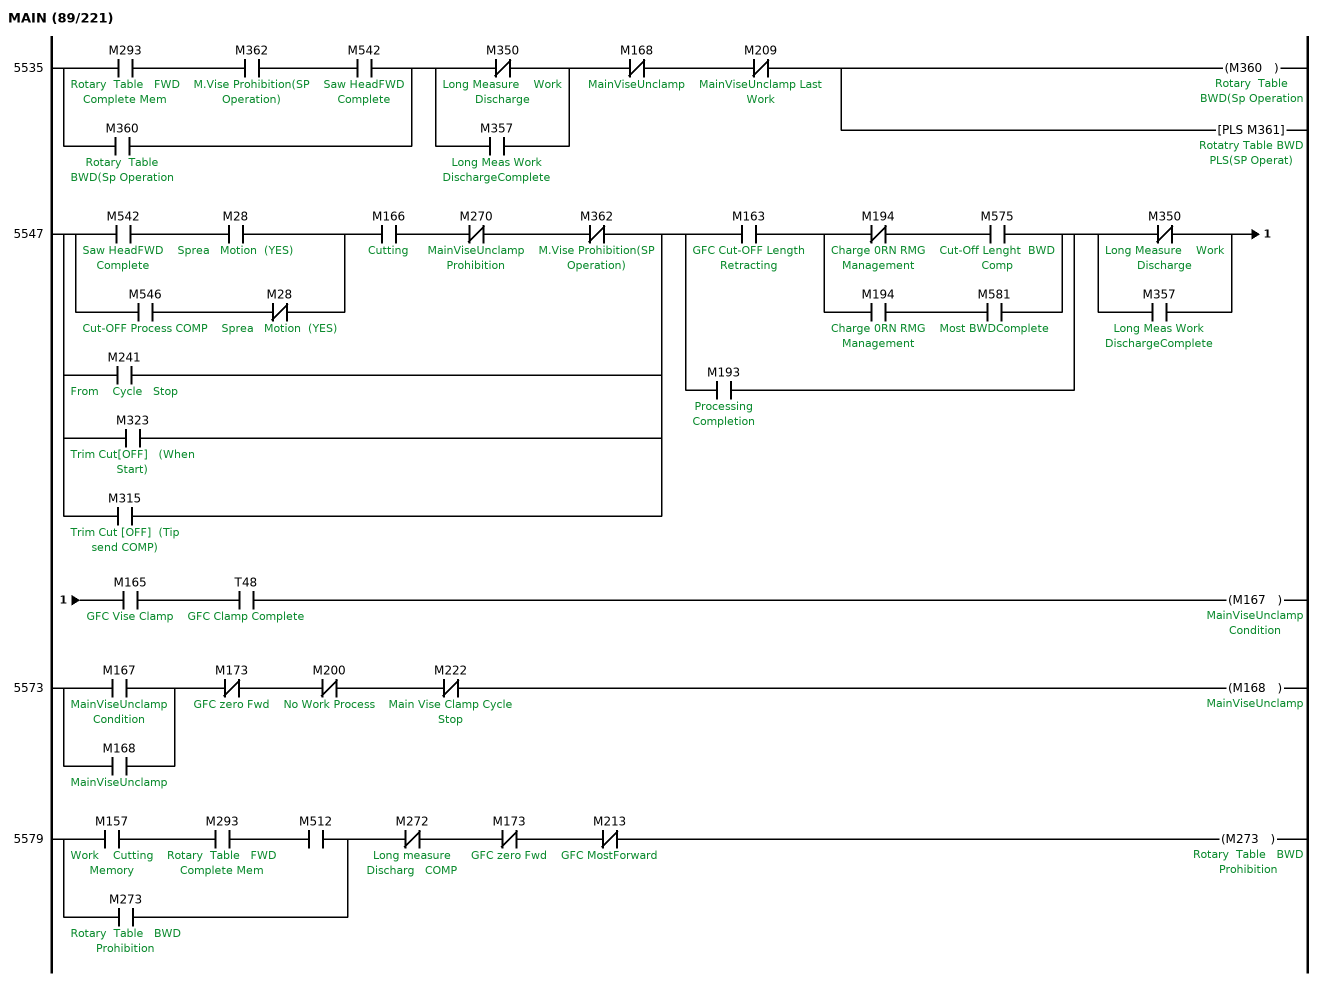
5535  LD      M293  ; Rotary  Table   FWD Complete Mem
      AND     M362  ; M.Vise Prohibition(SP Operation)
      AND     M542  ; Saw HeadFWD     Complete
      OR      M360  ; Rotary  Table   BWD(Sp Operation
      LDI     M350  ; Long Measure    Work Discharge
      OR      M357  ; Long Meas Work DischargeComplete
      ANB
      ANI     M168  ; MainViseUnclamp
      ANI     M209  ; MainViseUnclamp Last    Work
      OUT     M360  ; Rotary  Table   BWD(Sp Operation
      PLS     M361  ; Rotatry Table BWD PLS(SP Operat)
5547  LD      M542  ; Saw HeadFWD     Complete
      AND     M28  ; Sprea   Motion  (YES)
      LD      M546  ; Cut-OFF Process COMP
      ANI     M28  ; Sprea   Motion  (YES)
      ORB
      AND     M166  ; Cutting
      ANI     M270  ; MainViseUnclamp Prohibition
      ANI     M362  ; M.Vise Prohibition(SP Operation)
      OR      M241  ; From    Cycle   Stop
      OR      M323  ; Trim Cut[OFF]   (When   Start)
      OR      M315  ; Trim Cut [OFF]  (Tip send COMP)
      LD      M163  ; GFC Cut-OFF Length Retracting
      LDI     M194  ; Charge 0RN RMG  Management
      AND     M575  ; Cut-Off Lenght  BWD Comp
      LD      M194  ; Charge 0RN RMG  Management
      AND     M581  ; Most BWDComplete
      ORB
      ANB
      OR      M193  ; Processing      Completion
      ANB
      LDI     M350  ; Long Measure    Work Discharge
      OR      M357  ; Long Meas Work DischargeComplete
      ANB
      AND     M165  ; GFC Vise Clamp
      AND     T48  ; GFC Clamp Complete
      OUT     M167  ; MainViseUnclamp Condition
5573  LD      M167  ; MainViseUnclamp Condition
      OR      M168  ; MainViseUnclamp
      ANI     M173  ; GFC zero Fwd
      ANI     M200  ; No Work Process
      ANI     M222  ; Main Vise Clamp Cycle Stop
      OUT     M168  ; MainViseUnclamp
5579  LD      M157  ; Work    Cutting Memory
      AND     M293  ; Rotary  Table   FWD Complete Mem
      AND     M512
      OR      M273  ; Rotary  Table   BWD Prohibition
      ANI     M272  ; Long measure Discharg   COMP
      ANI     M173  ; GFC zero Fwd
      ANI     M213  ; GFC MostForward
      OUT     M273  ; Rotary  Table   BWD Prohibition
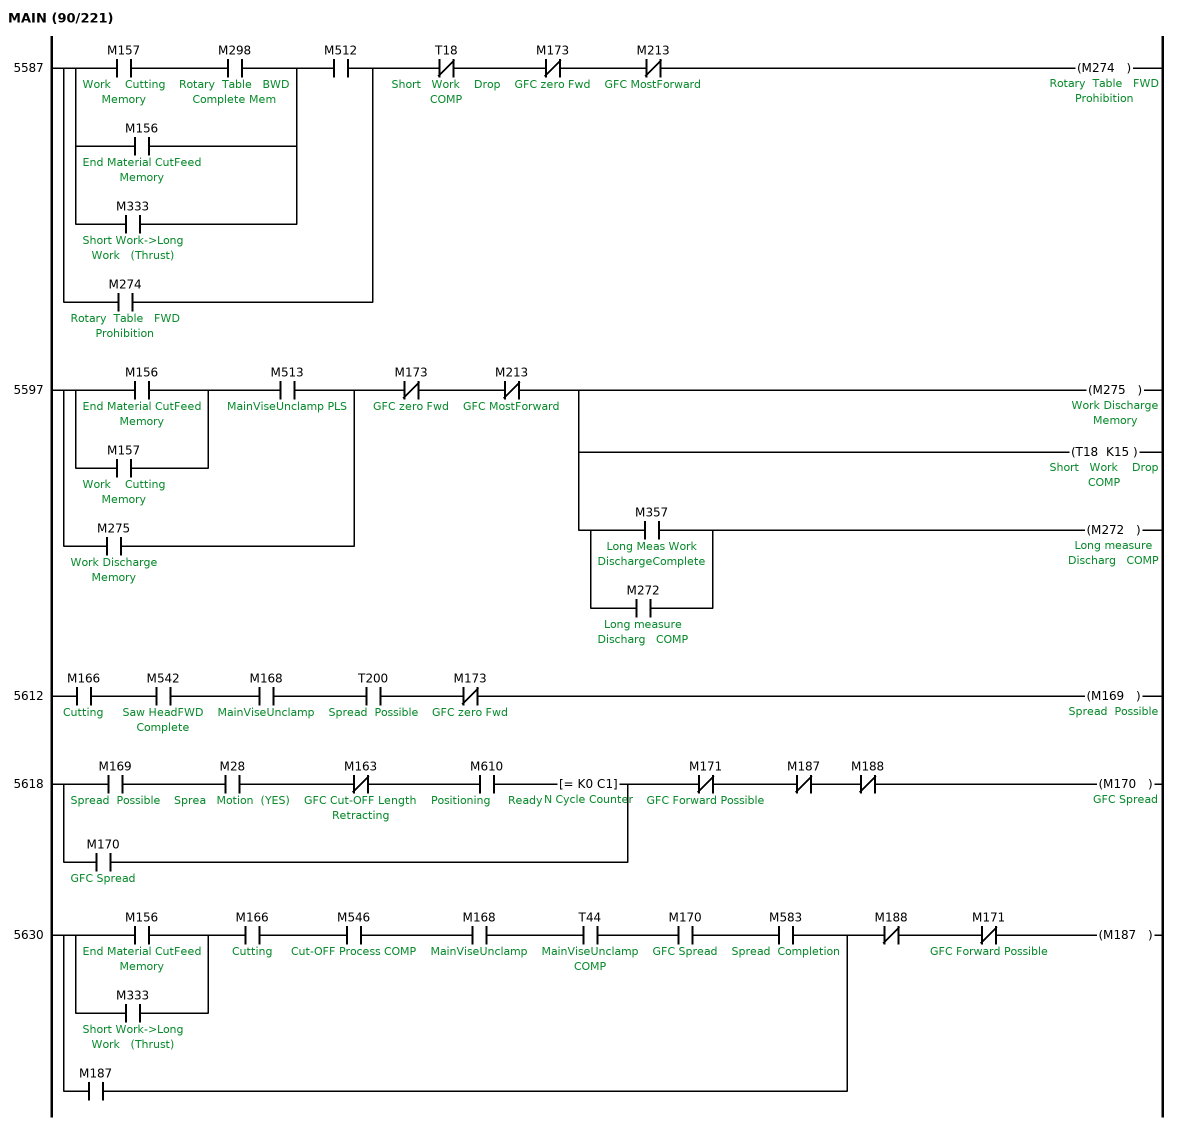
5587  LD      M157  ; Work    Cutting Memory
      AND     M298  ; Rotary  Table   BWD Complete Mem
      OR      M156  ; End Material CutFeed Memory
      OR      M333  ; Short Work->Long Work   (Thrust)
      AND     M512
      OR      M274  ; Rotary  Table   FWD Prohibition
      ANI     T18  ; Short   Work    Drop    COMP
      ANI     M173  ; GFC zero Fwd
      ANI     M213  ; GFC MostForward
      OUT     M274  ; Rotary  Table   FWD Prohibition
5597  LD      M156  ; End Material CutFeed Memory
      OR      M157  ; Work    Cutting Memory
      AND     M513  ; MainViseUnclamp PLS
      OR      M275  ; Work Discharge  Memory
      ANI     M173  ; GFC zero Fwd
      ANI     M213  ; GFC MostForward
      OUT     M275  ; Work Discharge  Memory
      OUT     T18 K15  ; Short   Work    Drop    COMP
      LD      M357  ; Long Meas Work DischargeComplete
      OR      M272  ; Long measure Discharg   COMP
      ANB
      OUT     M272  ; Long measure Discharg   COMP
5612  LD      M166  ; Cutting
      AND     M542  ; Saw HeadFWD     Complete
      AND     M168  ; MainViseUnclamp
      AND     T200  ; Spread  Possible
      ANI     M173  ; GFC zero Fwd
      OUT     M169  ; Spread  Possible
5618  LD      M169  ; Spread  Possible
      AND     M28  ; Sprea   Motion  (YES)
      ANI     M163  ; GFC Cut-OFF Length Retracting
      AND     M610  ; Positioning     Ready
      AND=    K0 C1  ; N Cycle Counter
      OR      M170  ; GFC Spread
      ANI     M171  ; GFC Forward Possible
      ANI     M187
      ANI     M188
      OUT     M170  ; GFC Spread
5630  LD      M156  ; End Material CutFeed Memory
      OR      M333  ; Short Work->Long Work   (Thrust)
      AND     M166  ; Cutting
      AND     M546  ; Cut-OFF Process COMP
      AND     M168  ; MainViseUnclamp
      AND     T44  ; MainViseUnclamp COMP
      AND     M170  ; GFC Spread
      AND     M583  ; Spread  Completion
      OR      M187
      ANI     M188
      ANI     M171  ; GFC Forward Possible
      OUT     M187
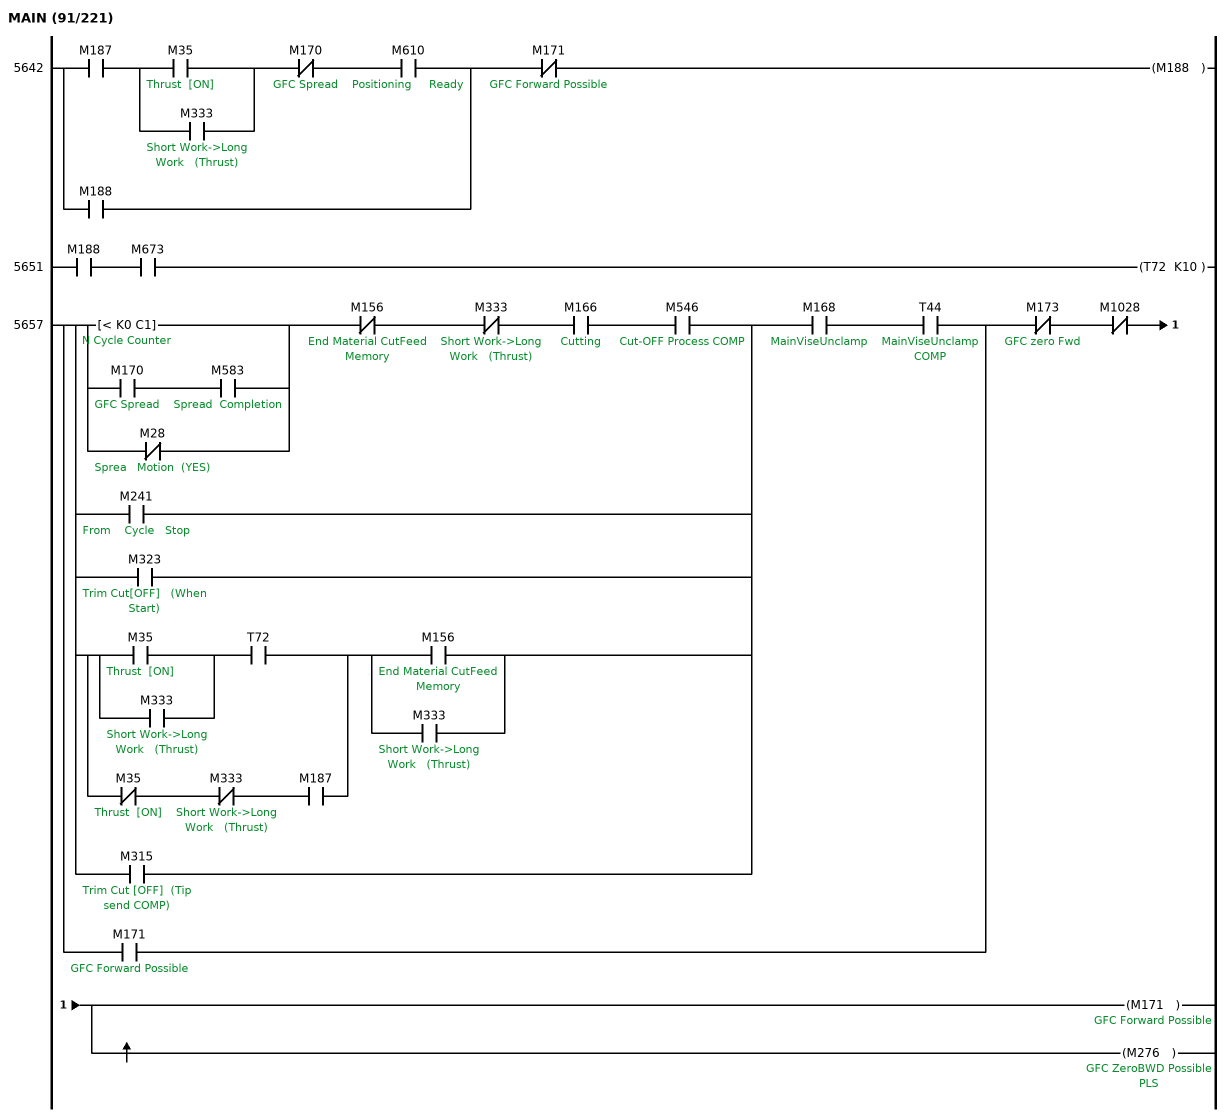
5642  LD      M187
      LD      M35  ; Thrust  [ON]
      OR      M333  ; Short Work->Long Work   (Thrust)
      ANB
      ANI     M170  ; GFC Spread
      AND     M610  ; Positioning     Ready
      OR      M188
      ANI     M171  ; GFC Forward Possible
      OUT     M188
5651  LD      M188
      AND     M673
      OUT     T72 K10
5657  LD<     K0 C1  ; N Cycle Counter
      LD      M170  ; GFC Spread
      AND     M583  ; Spread  Completion
      ORB
      ORI     M28  ; Sprea   Motion  (YES)
      ANI     M156  ; End Material CutFeed Memory
      ANI     M333  ; Short Work->Long Work   (Thrust)
      AND     M166  ; Cutting
      AND     M546  ; Cut-OFF Process COMP
      OR      M241  ; From    Cycle   Stop
      OR      M323  ; Trim Cut[OFF]   (When   Start)
      LD      M35  ; Thrust  [ON]
      OR      M333  ; Short Work->Long Work   (Thrust)
      AND     T72
      LDI     M35  ; Thrust  [ON]
      ANI     M333  ; Short Work->Long Work   (Thrust)
      AND     M187
      ORB
      LD      M156  ; End Material CutFeed Memory
      OR      M333  ; Short Work->Long Work   (Thrust)
      ANB
      ORB
      OR      M315  ; Trim Cut [OFF]  (Tip send COMP)
      AND     M168  ; MainViseUnclamp
      AND     T44  ; MainViseUnclamp COMP
      OR      M171  ; GFC Forward Possible
      ANI     M173  ; GFC zero Fwd
      ANI     M1028
      OUT     M171  ; GFC Forward Possible
      MEP
      OUT     M276  ; GFC ZeroBWD Possible PLS
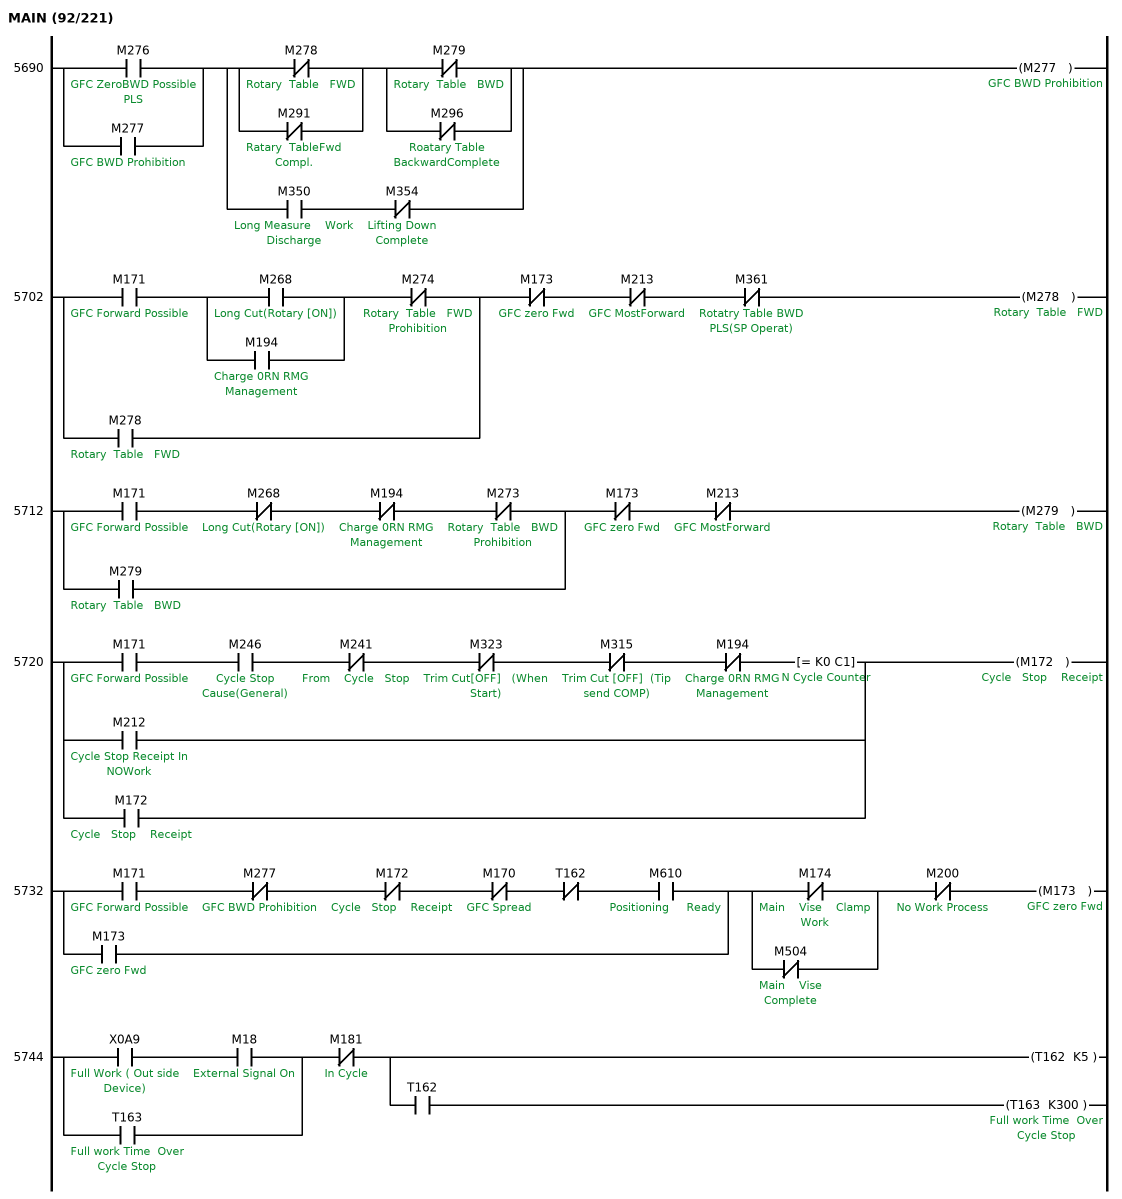
5690  LD      M276  ; GFC ZeroBWD Possible PLS
      OR      M277  ; GFC BWD Prohibition
      LDI     M278  ; Rotary  Table   FWD
      ORI     M291  ; Ratary  TableFwd Compl.
      LDI     M279  ; Rotary  Table   BWD
      ORI     M296  ; Roatary Table   BackwardComplete
      ANB
      LD      M350  ; Long Measure    Work Discharge
      ANI     M354  ; Lifting Down    Complete
      ORB
      ANB
      OUT     M277  ; GFC BWD Prohibition
5702  LD      M171  ; GFC Forward Possible
      LD      M268  ; Long Cut(Rotary [ON])
      OR      M194  ; Charge 0RN RMG  Management
      ANB
      ANI     M274  ; Rotary  Table   FWD Prohibition
      OR      M278  ; Rotary  Table   FWD
      ANI     M173  ; GFC zero Fwd
      ANI     M213  ; GFC MostForward
      ANI     M361  ; Rotatry Table BWD PLS(SP Operat)
      OUT     M278  ; Rotary  Table   FWD
5712  LD      M171  ; GFC Forward Possible
      ANI     M268  ; Long Cut(Rotary [ON])
      ANI     M194  ; Charge 0RN RMG  Management
      ANI     M273  ; Rotary  Table   BWD Prohibition
      OR      M279  ; Rotary  Table   BWD
      ANI     M173  ; GFC zero Fwd
      ANI     M213  ; GFC MostForward
      OUT     M279  ; Rotary  Table   BWD
5720  LD      M171  ; GFC Forward Possible
      AND     M246  ; Cycle Stop Cause(General)
      ANI     M241  ; From    Cycle   Stop
      ANI     M323  ; Trim Cut[OFF]   (When   Start)
      ANI     M315  ; Trim Cut [OFF]  (Tip send COMP)
      ANI     M194  ; Charge 0RN RMG  Management
      AND=    K0 C1  ; N Cycle Counter
      OR      M212  ; Cycle Stop Receipt In NOWork
      OR      M172  ; Cycle   Stop    Receipt
      OUT     M172  ; Cycle   Stop    Receipt
5732  LD      M171  ; GFC Forward Possible
      ANI     M277  ; GFC BWD Prohibition
      ANI     M172  ; Cycle   Stop    Receipt
      ANI     M170  ; GFC Spread
      ANI     T162
      AND     M610  ; Positioning     Ready
      OR      M173  ; GFC zero Fwd
      LDI     M174  ; Main    Vise    Clamp   Work
      ORI     M504  ; Main    Vise    Complete
      ANB
      ANI     M200  ; No Work Process
      OUT     M173  ; GFC zero Fwd
5744  LD      X0A9  ; Full Work ( Out side Device)
      AND     M18  ; External Signal On
      OR      T163  ; Full work Time  Over Cycle Stop
      ANI     M181  ; In Cycle
      OUT     T162 K5
      AND     T162
      OUT     T163 K300  ; Full work Time  Over Cycle Stop
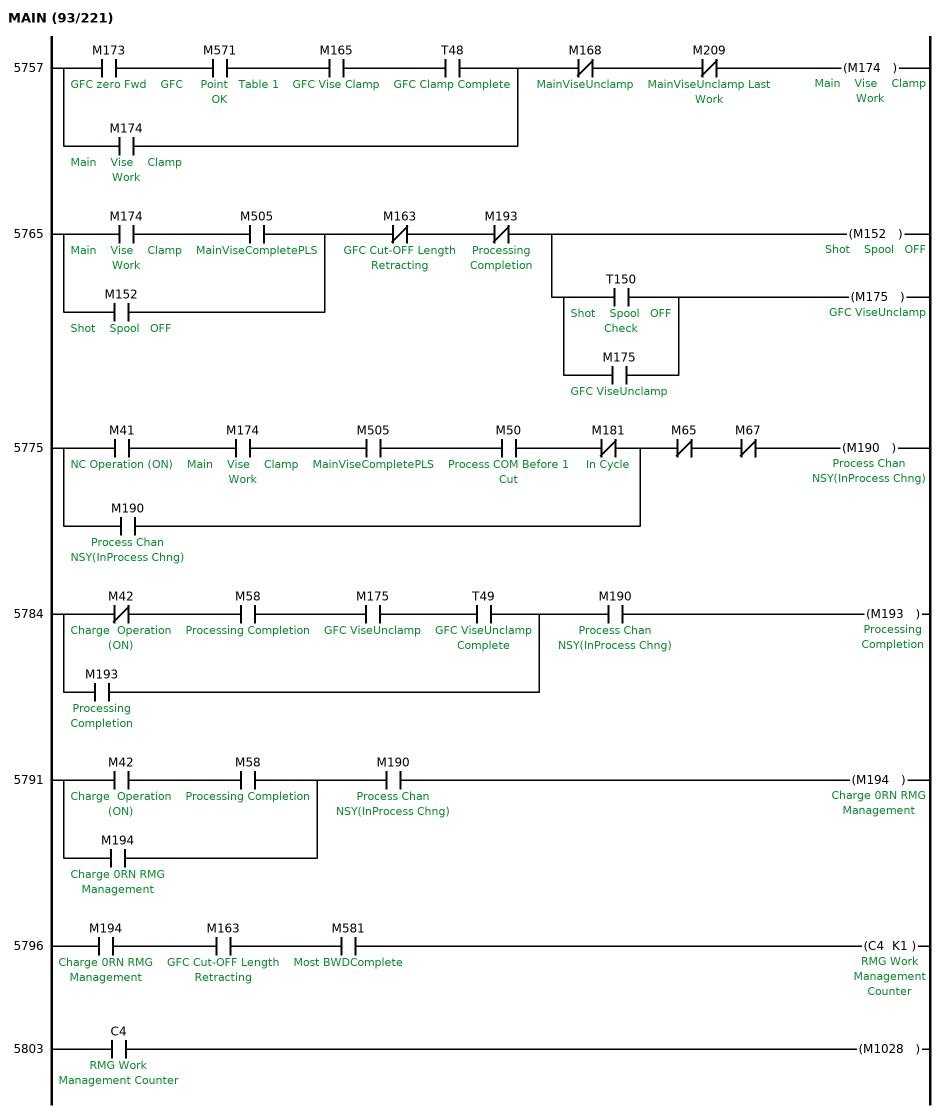
5757  LD      M173  ; GFC zero Fwd
      AND     M571  ; GFC     Point   Table 1 OK
      AND     M165  ; GFC Vise Clamp
      AND     T48  ; GFC Clamp Complete
      OR      M174  ; Main    Vise    Clamp   Work
      ANI     M168  ; MainViseUnclamp
      ANI     M209  ; MainViseUnclamp Last    Work
      OUT     M174  ; Main    Vise    Clamp   Work
5765  LD      M174  ; Main    Vise    Clamp   Work
      AND     M505  ; MainViseCompletePLS
      OR      M152  ; Shot    Spool   OFF
      ANI     M163  ; GFC Cut-OFF Length Retracting
      ANI     M193  ; Processing      Completion
      OUT     M152  ; Shot    Spool   OFF
      LD      T150  ; Shot    Spool   OFF     Check
      OR      M175  ; GFC ViseUnclamp
      ANB
      OUT     M175  ; GFC ViseUnclamp
5775  LD      M41  ; NC Operation (ON)
      AND     M174  ; Main    Vise    Clamp   Work
      AND     M505  ; MainViseCompletePLS
      AND     M50  ; Process COM Before 1 Cut
      ANI     M181  ; In Cycle
      OR      M190  ; Process Chan NSY(InProcess Chng)
      ANI     M65
      ANI     M67
      OUT     M190  ; Process Chan NSY(InProcess Chng)
5784  LDI     M42  ; Charge  Operation (ON)
      AND     M58  ; Processing Completion
      AND     M175  ; GFC ViseUnclamp
      AND     T49  ; GFC ViseUnclamp Complete
      OR      M193  ; Processing      Completion
      AND     M190  ; Process Chan NSY(InProcess Chng)
      OUT     M193  ; Processing      Completion
5791  LD      M42  ; Charge  Operation (ON)
      AND     M58  ; Processing Completion
      OR      M194  ; Charge 0RN RMG  Management
      AND     M190  ; Process Chan NSY(InProcess Chng)
      OUT     M194  ; Charge 0RN RMG  Management
5796  LD      M194  ; Charge 0RN RMG  Management
      AND     M163  ; GFC Cut-OFF Length Retracting
      AND     M581  ; Most BWDComplete
      OUT     C4 K1  ; RMG WorkManagement Counter
5803  LD      C4  ; RMG WorkManagement Counter
      OUT     M1028
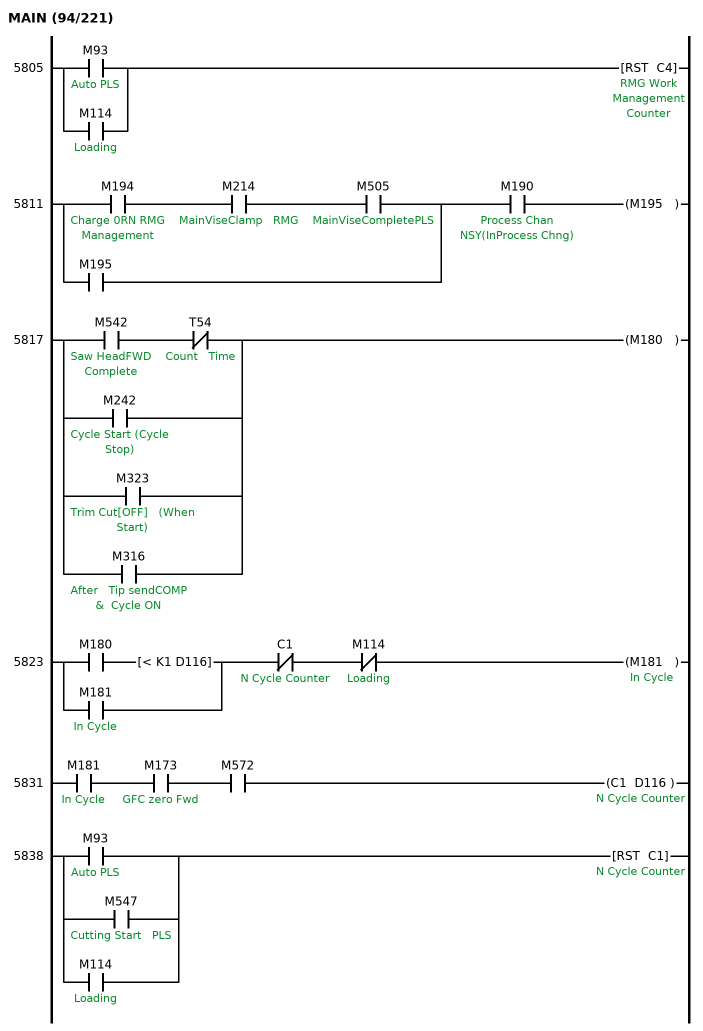
5805  LD      M93  ; Auto PLS
      OR      M114  ; Loading
      RST     C4  ; RMG WorkManagement Counter
5811  LD      M194  ; Charge 0RN RMG  Management
      AND     M214  ; MainViseClamp   RMG
      AND     M505  ; MainViseCompletePLS
      OR      M195
      AND     M190  ; Process Chan NSY(InProcess Chng)
      OUT     M195
5817  LD      M542  ; Saw HeadFWD     Complete
      ANI     T54  ; Count   Time
      OR      M242  ; Cycle Start (Cycle Stop)
      OR      M323  ; Trim Cut[OFF]   (When   Start)
      OR      M316  ; After   Tip sendCOMP &  Cycle ON
      OUT     M180
5823  LD      M180
      AND<    K1 D116
      OR      M181  ; In Cycle
      ANI     C1  ; N Cycle Counter
      ANI     M114  ; Loading
      OUT     M181  ; In Cycle
5831  LD      M181  ; In Cycle
      AND     M173  ; GFC zero Fwd
      AND     M572
      OUT     C1 D116  ; N Cycle Counter
5838  LD      M93  ; Auto PLS
      OR      M547  ; Cutting Start   PLS
      OR      M114  ; Loading
      RST     C1  ; N Cycle Counter
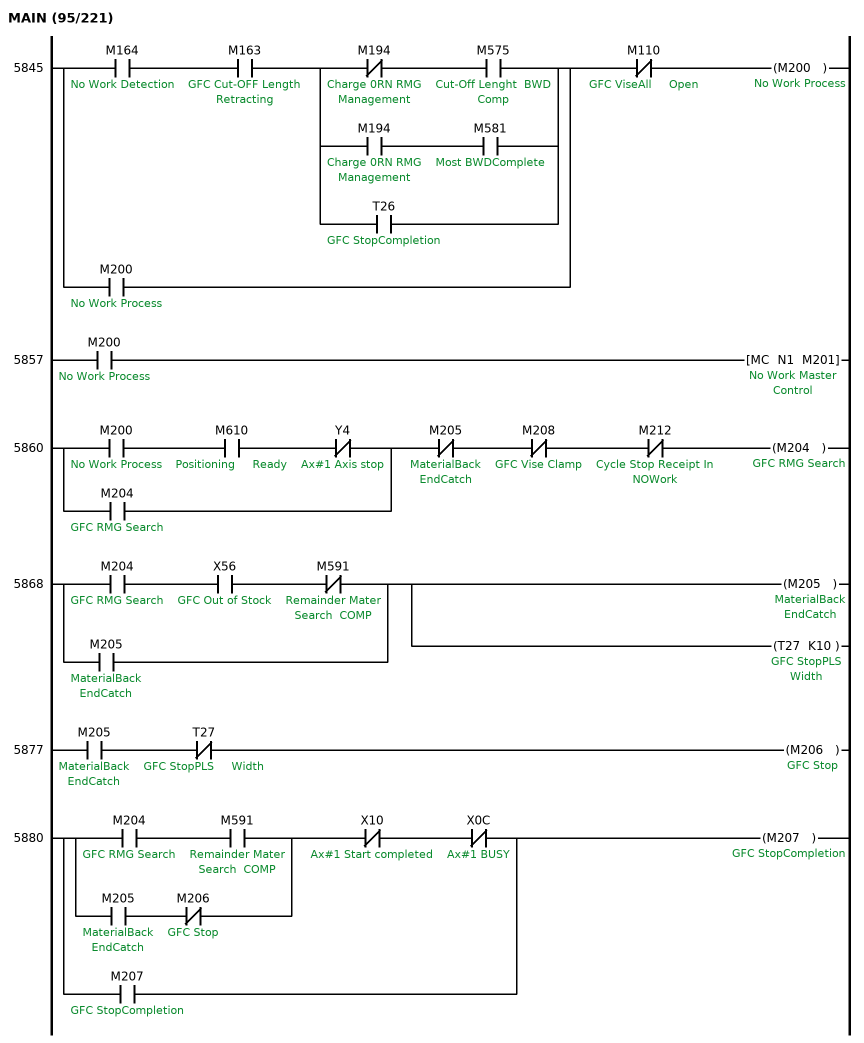
5845  LD      M164  ; No Work Detection
      AND     M163  ; GFC Cut-OFF Length Retracting
      LDI     M194  ; Charge 0RN RMG  Management
      AND     M575  ; Cut-Off Lenght  BWD Comp
      LD      M194  ; Charge 0RN RMG  Management
      AND     M581  ; Most BWDComplete
      ORB
      OR      T26  ; GFC StopCompletion
      ANB
      OR      M200  ; No Work Process
      ANI     M110  ; GFC ViseAll     Open
      OUT     M200  ; No Work Process
5857  LD      M200  ; No Work Process
      MC      N1 M201  ; No Work Master  Control
5860  LD      M200  ; No Work Process
      AND     M610  ; Positioning     Ready
      ANI     Y4  ; Ax#1 Axis stop
      OR      M204  ; GFC RMG Search
      ANI     M205  ; MaterialBack EndCatch
      ANI     M208  ; GFC Vise Clamp
      ANI     M212  ; Cycle Stop Receipt In NOWork
      OUT     M204  ; GFC RMG Search
5868  LD      M204  ; GFC RMG Search
      AND     X56  ; GFC Out of Stock
      ANI     M591  ; Remainder Mater Search  COMP
      OR      M205  ; MaterialBack EndCatch
      OUT     M205  ; MaterialBack EndCatch
      OUT     T27 K10  ; GFC StopPLS     Width
5877  LD      M205  ; MaterialBack EndCatch
      ANI     T27  ; GFC StopPLS     Width
      OUT     M206  ; GFC Stop
5880  LD      M204  ; GFC RMG Search
      AND     M591  ; Remainder Mater Search  COMP
      LD      M205  ; MaterialBack EndCatch
      ANI     M206  ; GFC Stop
      ORB
      ANI     X10  ; Ax#1 Start completed
      ANI     X0C  ; Ax#1 BUSY
      OR      M207  ; GFC StopCompletion
      OUT     M207  ; GFC StopCompletion
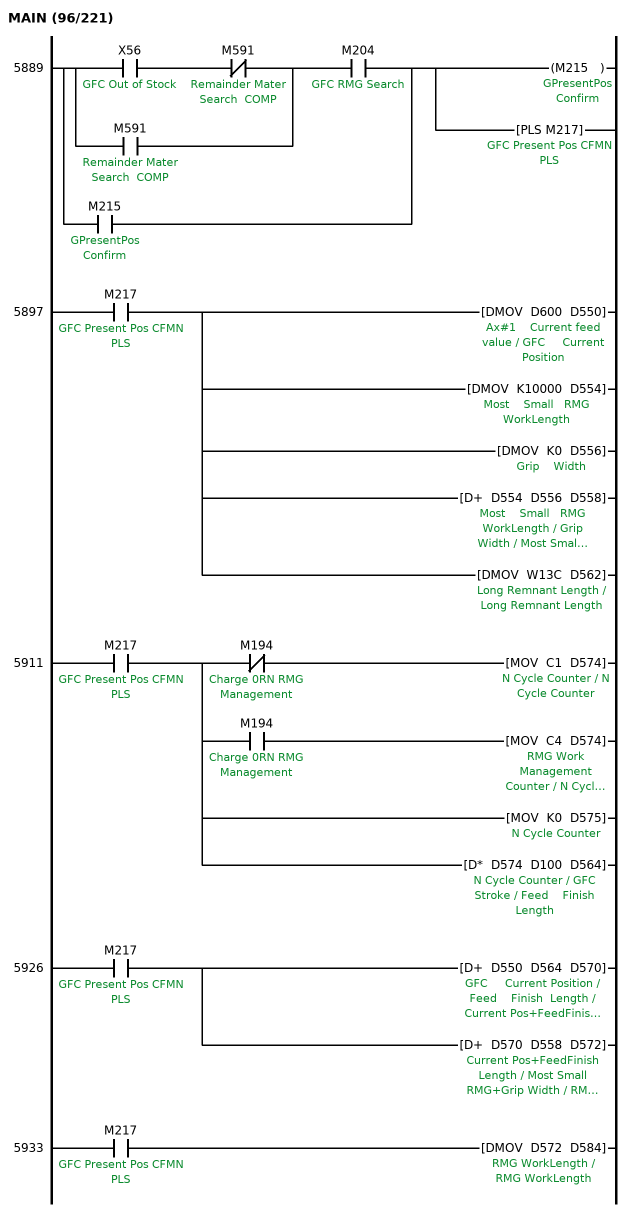
5889  LD      X56  ; GFC Out of Stock
      ANI     M591  ; Remainder Mater Search  COMP
      OR      M591  ; Remainder Mater Search  COMP
      AND     M204  ; GFC RMG Search
      OR      M215  ; GPresentPos     Confirm
      OUT     M215  ; GPresentPos     Confirm
      PLS     M217  ; GFC Present Pos CFMN PLS
5897  LD      M217  ; GFC Present Pos CFMN PLS
      DMOV    D600 D550  ; GFC     Current Position
      DMOV    K10000 D554  ; Most    Small   RMG WorkLength
      DMOV    K0 D556  ; Grip    Width
      D+      D554 D556 D558  ; Most Small RMG+Grip Width
      DMOV    W13C D562  ; Long Remnant Length / Long Remnant Length
5911  LD      M217  ; GFC Present Pos CFMN PLS
      MPS
      ANI     M194  ; Charge 0RN RMG  Management
      MOV     C1 D574  ; N Cycle Counter
      MRD
      AND     M194  ; Charge 0RN RMG  Management
      MOV     C4 D574
      MPP
      MOV     K0 D575  ; N Cycle Counter
      D*      D574 D100 D564  ; GFC     Stroke / Feed    Finish  Length
5926  LD      M217  ; GFC Present Pos CFMN PLS
      D+      D550 D564 D570  ; Current Pos+FeedFinish  Length
      D+      D570 D558 D572  ; RMG WorkLength
5933  LD      M217  ; GFC Present Pos CFMN PLS
      DMOV    D572 D584  ; RMG WorkLength
